# B&R Automation Studio project TD52 (part 76)

#### lib_properties.txt
```
For manual assignment to hardware configuration please
add the following additional include directories:

\Logical\MATLAB_includes\R2012b\

And the following additional build options:

-lm -D MODEL=LX2 -D NUMST=1 -D NCSTATES=0 -D HAVESTDIO -D ONESTEPFCN=1 -D TERMFCN=1 -D MAT_FILE=0 -D MULTI_INSTANCE_CODE=0 -D INTEGER_CODE=0 -D MT=0 -D CLASSIC_INTERFACE=0 -D TID01EQ=0
```

### Library Logical/EngineController/Lib_EC/lDAI (ANSIC, version 1.00.0) - Direct Air Injection 

#### DAI.c
```c
/********************************************************************
 * COPYRIGHT -- B&R Industrial Automation GmbH
 ********************************************************************
 * Program: DAI
 * File: DAI.c
 * Author: 105055527
 * Last modified by: cadm_kafkama00
 * Created: Sat Nov 11 23:05:34 2017
 * Last modified: Wed Oct 02 14:21:06 2024
 * Model Version: 4.14
 * Description: Direct Air Injection for J920 Faststart

   History:

   V0.02  Arnold, 27.11.2017,  tech demonstrator @ P20
   V0.03  Arnold, 24.10.2018,  rename from AirAss to DAI
   V0.04  Arnold, 24.10.2018,  deleted exhaust side DAI, deleted intake dynamics
   V0.05  Arnold, 14.08.2019,  unit testing done, pre-release for Pforzheim P21
   V0.06  Kafka, 20.09.2019, bug fix for testbench manual massflow testing
   V0.07  Kafka, 01.10.2019, massflow limitations changed from per valve to total massflow
   V0.08  Kafka, 02.10.2019, mass flow limitation over boost pressure removed for speed ramp
   V0.09  Kafka, 14.10.2019, disable for negative power trajectory is added in the enable subblock
   V0.10  Kafka, 18.12.2019, disable on speed hysteresis during speed ramp
   V4.14  Kafka, 06.09.2024, update to Matlab Version 2021b

 * modified Comment:
 ********************************************************************
 * Implementation of program DAI
 ********************************************************************
 * Generated with B&R Automation Studio Target for Simulink V6.7.1
 * (ERT based)
 ********************************************************************/

#include "DAI.h"
#include "DAI_private.h"

/*  Defines */

/*  Data Types */

/**************************** GLOBAL DATA *************************************/
/*  Definitions */

/*  Declarations  */

/* Forward declaration for local functions */
static void DAI_merge(int32_T idx[5], real32_T x[5], int32_T offset, int32_T np,
                      int32_T nq, int32_T iwork[5], real32_T xwork[5], struct fDAI* inst);
static void DAI_sort(real32_T x[5], int32_T idx[5], struct fDAI* inst);

/***************************** FILE SCOPE DATA ********************************/

/*************************** FUNCTIONS ****************************************/

/* Lookup Binary Search Utility BINARYSEARCH_real32_T */
void BINARYSEARCH_real32_T(uint32_T *piLeft, uint32_T *piRght, real32_T u, const
  real32_T *pData, uint32_T iHi, struct fDAI* inst)
{
  /* Find the location of current input value in the data table. */
  *piLeft = 0U;
  *piRght = iHi;
  if (u <= pData[0] ) {
    /* Less than or equal to the smallest point in the table. */
    *piRght = 0U;
  } else if (u >= pData[iHi] ) {
    /* Greater than or equal to the largest point in the table. */
    *piLeft = iHi;
  } else {
    uint32_T i;

    /* Do a binary search. */
    while (( *piRght - *piLeft ) > 1U ) {
      /* Get the average of the left and right indices using to Floor rounding. */
      i = (*piLeft + *piRght) >> 1;

      /* Move either the right index or the left index so that */
      /*  LeftDataPoint <= CurrentValue < RightDataPoint */
      if (u < pData[i] ) {
        *piRght = i;
      } else {
        *piLeft = i;
      }
    }
  }
}

/* Lookup Utility LookUp_real32_T_real32_T */
void LookUp_real32_T_real32_T(real32_T *pY, const real32_T *pYData, real32_T u,
  const real32_T *pUData, uint32_T iHi, struct fDAI* inst)
{
  uint32_T iLeft;
  uint32_T iRght;
  BINARYSEARCH_real32_T( &(iLeft), &(iRght), u, pUData, iHi, inst);

  {
    real32_T lambda;
    if (pUData[iRght] > pUData[iLeft] ) {
      real32_T num;
      real32_T den;
      den = pUData[iRght];
      den -= pUData[iLeft];
      num = u;
      num -= pUData[iLeft];
      lambda = num / den;
    } else {
      lambda = 0.0F;
    }

    {
      real32_T yLeftCast;
      real32_T yRghtCast;
      yLeftCast = pYData[iLeft];
      yRghtCast = pYData[iRght];
      yLeftCast += lambda * ( yRghtCast - yLeftCast );
      (*pY) = yLeftCast;
    }
  }
}

/*
 * Output and update for atomic system:
 *    '<S2>/Hystersis'
 *    '<S2>/Hystersis2'
 */
void DAI_Hystersis(real32_T rtu_Gw, real32_T rtu_Hy, real32_T rtu_In,
                   rtB_Hystersis_DAI *localB, rtDW_Hystersis_DAI *localDW, struct fDAI* inst)
{
  localDW->Inter = ((rtu_In >= rtu_Gw) || ((rtu_In >= rtu_Gw - rtu_Hy) &&
    localDW->Inter));
  localB->Out = localDW->Inter;
}

/* Function for MATLAB Function: '<S10>/MATLAB Function' */
static void DAI_merge(int32_T idx[5], real32_T x[5], int32_T offset, int32_T np,
                      int32_T nq, int32_T iwork[5], real32_T xwork[5], struct fDAI* inst)
{
  int32_T q;
  if ((np != 0) && (nq != 0)) {
    int32_T iout;
    int32_T n;
    int32_T n_tmp;
    n_tmp = np + nq;
    for (q = 0; q < n_tmp; q++) {
      iout = offset + q;
      iwork[q] = idx[iout];
      xwork[q] = x[iout];
    }

    n = 0;
    q = np;
    iout = offset - 1;
    int32_T exitg1;
    do {
      exitg1 = 0;
      iout++;
      if (xwork[n] <= xwork[q]) {
        idx[iout] = iwork[n];
        x[iout] = xwork[n];
        if (n + 1 < np) {
          n++;
        } else {
          exitg1 = 1;
        }
      } else {
        idx[iout] = iwork[q];
        x[iout] = xwork[q];
        if (q + 1 < n_tmp) {
          q++;
        } else {
          q = iout - n;
          while (n + 1 <= np) {
            iout = (q + n) + 1;
            idx[iout] = iwork[n];
            x[iout] = xwork[n];
            n++;
          }

          exitg1 = 1;
        }
      }
    } while (exitg1 == 0);
  }
}

/* Function for MATLAB Function: '<S10>/MATLAB Function' */
static void DAI_sort(real32_T x[5], int32_T idx[5], struct fDAI* inst)
{
  int32_T iwork[5];
  int32_T i2;
  int32_T i3;
  int32_T ib;
  int32_T k;
  real32_T xwork[5];
  real32_T x4[4];
  int8_T idx4[4];
  int8_T perm[4];
  x4[0] = 0.0F;
  idx4[0] = 0;
  x4[1] = 0.0F;
  idx4[1] = 0;
  x4[2] = 0.0F;
  idx4[2] = 0;
  x4[3] = 0.0F;
  idx4[3] = 0;
  ib = 0;
  for (k = 0; k < 5; k++) {
    idx[k] = 0;
    ib++;
    idx4[ib - 1] = (int8_T)(k + 1);
    x4[ib - 1] = x[k];
    if (ib == 4) {
      int32_T i4;
      real32_T tmp;
      real32_T tmp_0;
      if (x4[0] <= x4[1]) {
        ib = 1;
        i2 = 2;
      } else {
        ib = 2;
        i2 = 1;
      }

      if (x4[2] <= x4[3]) {
        i3 = 3;
        i4 = 4;
      } else {
        i3 = 4;
        i4 = 3;
      }

      tmp = x4[ib - 1];
      tmp_0 = x4[i3 - 1];
      if (tmp <= tmp_0) {
        tmp = x4[i2 - 1];
        if (tmp <= tmp_0) {
          perm[0] = (int8_T)ib;
          perm[1] = (int8_T)i2;
          perm[2] = (int8_T)i3;
          perm[3] = (int8_T)i4;
        } else if (tmp <= x4[i4 - 1]) {
          perm[0] = (int8_T)ib;
          perm[1] = (int8_T)i3;
          perm[2] = (int8_T)i2;
          perm[3] = (int8_T)i4;
        } else {
          perm[0] = (int8_T)ib;
          perm[1] = (int8_T)i3;
          perm[2] = (int8_T)i4;
          perm[3] = (int8_T)i2;
        }
      } else {
        tmp_0 = x4[i4 - 1];
        if (tmp <= tmp_0) {
          if (x4[i2 - 1] <= tmp_0) {
            perm[0] = (int8_T)i3;
            perm[1] = (int8_T)ib;
            perm[2] = (int8_T)i2;
            perm[3] = (int8_T)i4;
          } else {
            perm[0] = (int8_T)i3;
            perm[1] = (int8_T)ib;
            perm[2] = (int8_T)i4;
            perm[3] = (int8_T)i2;
          }
        } else {
          perm[0] = (int8_T)i3;
          perm[1] = (int8_T)i4;
          perm[2] = (int8_T)ib;
          perm[3] = (int8_T)i2;
        }
      }

      idx[k - 3] = idx4[perm[0] - 1];
      idx[k - 2] = idx4[perm[1] - 1];
      idx[k - 1] = idx4[perm[2] - 1];
      idx[k] = idx4[perm[3] - 1];
      x[k - 3] = x4[perm[0] - 1];
      x[k - 2] = x4[perm[1] - 1];
      x[k - 1] = x4[perm[2] - 1];
      x[k] = x4[perm[3] - 1];
      ib = 0;
    }
  }

  if (ib > 0) {
    perm[1] = 0;
    perm[2] = 0;
    perm[3] = 0;
    if (ib == 1) {
      perm[0] = 1;
    } else if (ib == 2) {
      if (x4[0] <= x4[1]) {
        perm[0] = 1;
        perm[1] = 2;
      } else {
        perm[0] = 2;
        perm[1] = 1;
      }
    } else if (x4[0] <= x4[1]) {
      if (x4[1] <= x4[2]) {
        perm[0] = 1;
        perm[1] = 2;
        perm[2] = 3;
      } else if (x4[0] <= x4[2]) {
        perm[0] = 1;
        perm[1] = 3;
        perm[2] = 2;
      } else {
        perm[0] = 3;
        perm[1] = 1;
        perm[2] = 2;
      }
    } else if (x4[0] <= x4[2]) {
      perm[0] = 2;
      perm[1] = 1;
      perm[2] = 3;
    } else if (x4[1] <= x4[2]) {
      perm[0] = 2;
      perm[1] = 3;
      perm[2] = 1;
    } else {
      perm[0] = 3;
      perm[1] = 2;
      perm[2] = 1;
    }

    for (k = 0; k < ib; k++) {
      i2 = perm[k] - 1;
      i3 = (k - ib) + 5;
      idx[i3] = idx4[i2];
      x[i3] = x4[i2];
    }
  }

  for (k = 0; k < 5; k++) {
    iwork[k] = 0;
    xwork[k] = 0.0F;
  }

  DAI_merge(idx, x, 0, 4, 1, iwork, xwork, inst);
}

/* Model step function */
void DAI_step(RT_MODEL_DAI *const DAI_M, struct fDAI* inst)
{
  struct BlockIO_DAI *DAI_B = DAI_M->blockIO;
  struct D_Work_DAI *DAI_DWork = DAI_M->dwork;

  /* local block i/o variables */
  real32_T rtb_CorrInternal[2];
  real32_T rtb_LookupTableDynamic2;
  real32_T rtb_LookupTableDynamic2_g;
  real32_T rtb_Saturation2[2];
  int32_T iidx[5];
  int32_T i;
  real32_T rtb_x_out[5];
  real32_T rtb_y_out[5];
  real32_T rtb_rCd[2];
  real32_T rtb_Disableintakedynamics1;
  real32_T rtb_Product_nc;
  real32_T rtb_Switch2_i;
  real32_T rtb_Switch2_n;
  real32_T rtb_UkYk1;
  real32_T rtb_rFlow_eng_act;
  real32_T rtb_rFlow_eng_des;
  boolean_T rtb_LogicalOperator2;
  boolean_T rtb_LogicalOperator5;

  /* S-Function (bur_bus_in): '<Root>/Bus Input3' */
  DAI_B->BusInput3 = inst->In;

  /* S-Function (bur_bus_in): '<Root>/Bus Input1' */
  DAI_B->BusInput1 = inst->Para;

  /* Outputs for Atomic SubSystem: '<Root>/EngineMassFlow' */
  /* MATLAB Function: '<S3>/desired engine massflow' incorporates:
   *  Constant: '<S27>/Constant1'
   *  MATLAB Function: '<S3>/actual engine massflow'
   *  Sum: '<S27>/Add1'
   */
  rtb_rFlow_eng_act = fmaxf((DAI_B->BusInput3.rT_T2s + 273.15F) * 287.15F, 1.0F);
  rtb_Disableintakedynamics1 = DAI_B->BusInput3.rVE_Eng *
    DAI_B->BusInput3.rV_EngDis;

  /* Outputs for Atomic SubSystem: '<Root>/Enable' */
  /* Product: '<S3>/Product' incorporates:
   *  Product: '<S2>/Product'
   */
  rtb_Product_nc = DAI_B->BusInput3.rN_Set_Norm * DAI_B->BusInput1.rN_EngNom;

  /* End of Outputs for SubSystem: '<Root>/Enable' */

  /* MATLAB Function: '<S3>/desired engine massflow' incorporates:
   *  Constant: '<S25>/Constant1'
   *  Constant: '<S30>/Constant1'
   *  Product: '<S25>/Product'
   *  Product: '<S30>/Product'
   *  Product: '<S3>/Product'
   */
  rtb_rFlow_eng_des = DAI_B->BusInput3.rPr_P2s_des * 100000.0F *
    rtb_Disableintakedynamics1 / rtb_rFlow_eng_act * (rtb_Product_nc *
    0.104719758F) / 2.0F / 6.28318548F;

  /* Switch: '<S23>/Switch2' incorporates:
   *  Constant: '<S3>/Constant4'
   *  RelationalOperator: '<S23>/LowerRelop1'
   *  RelationalOperator: '<S23>/UpperRelop'
   *  Switch: '<S23>/Switch'
   */
  if (DAI_B->BusInput3.rN_Eng > DAI_B->BusInput1.rN_EngNom) {
    rtb_Switch2_i = DAI_B->BusInput1.rN_EngNom;
  } else if (DAI_B->BusInput3.rN_Eng < 1.0F) {
    /* Switch: '<S23>/Switch' incorporates:
     *  Constant: '<S3>/Constant4'
     */
    rtb_Switch2_i = 1.0F;
  } else {
    rtb_Switch2_i = DAI_B->BusInput3.rN_Eng;
  }

  /* End of Switch: '<S23>/Switch2' */

  /* MATLAB Function: '<S3>/actual engine massflow' incorporates:
   *  Constant: '<S26>/Constant1'
   *  Constant: '<S29>/Constant1'
   *  Product: '<S26>/Product'
   *  Product: '<S29>/Product'
   */
  rtb_rFlow_eng_act = DAI_B->BusInput3.rPr_P2s_Avg * 100000.0F *
    rtb_Disableintakedynamics1 / rtb_rFlow_eng_act * (rtb_Switch2_i *
    0.104719758F) / 2.0F / 6.28318548F;

  /* End of Outputs for SubSystem: '<Root>/EngineMassFlow' */

  /* S-Function (bur_bus_in): '<Root>/Bus Input2' */
  DAI_B->BusInput2 = inst->Perm;

  /* Outputs for Atomic SubSystem: '<Root>/AirFlowDemand' */
  /* MATLAB Function: '<S10>/MATLAB Function' incorporates:
   *  Product: '<S10>/Divide'
   *  SignalConversion generated from: '<S13>/ SFunction '
   */
  rtb_x_out[0] = DAI_B->BusInput1.rN_DAI_On;
  rtb_x_out[1] = DAI_B->BusInput1.rN_EngNom * DAI_B->BusInput2.rNref_ff[0];
  rtb_x_out[2] = DAI_B->BusInput1.rN_EngNom * DAI_B->BusInput2.rNref_ff[1];
  rtb_x_out[3] = DAI_B->BusInput1.rN_EngNom * DAI_B->BusInput2.rNref_ff[2];
  rtb_x_out[4] = DAI_B->BusInput1.rN_DAI_Off;
  DAI_sort(rtb_x_out, iidx, inst);
  for (i = 0; i < 5; i++) {
    rtb_y_out[i] = DAI_B->BusInput2.rFlowRef_ff[iidx[i] - 1];
  }

  /* End of MATLAB Function: '<S10>/MATLAB Function' */

  /* Switch: '<S1>/ManMode' incorporates:
   *  Constant: '<S22>/Constant'
   *  Constant: '<S6>/Constant'
   *  RelationalOperator: '<S22>/Compare'
   *  RelationalOperator: '<S6>/Compare'
   *  Switch: '<S1>/OpMode'
   *  Switch: '<S3>/Disable intake dynamics1'
   */
  if (DAI_B->BusInput3.Test.bManEnable) {
    rtb_Disableintakedynamics1 = DAI_B->BusInput3.Test.rManMassReq;
  } else if (DAI_B->BusInput3.iOpMode <= 45) {
    /* S-Function (sfix_look1_dyn): '<S10>/Lookup Table Dynamic2' incorporates:
     *  Switch: '<S1>/OpMode'
     */
    /* Dynamic Look-Up Table Block: '<S10>/Lookup Table Dynamic2'
     * Input0  Data Type:  Floating Point real32_T
     * Input1  Data Type:  Floating Point real32_T
     * Input2  Data Type:  Floating Point real32_T
     * Output0 Data Type:  Floating Point real32_T
     * Lookup Method: Linear_Endpoint
     *
     */
    LookUp_real32_T_real32_T( &(rtb_LookupTableDynamic2_g), &rtb_y_out[0],
      DAI_B->BusInput3.rN_Eng, &rtb_x_out[0], 4U, inst);

    /* Switch: '<S1>/OpMode' incorporates:
     *  Product: '<S10>/Product3'
     */
    rtb_Disableintakedynamics1 = DAI_B->BusInput1.rGain_DAI_Start *
      rtb_LookupTableDynamic2_g;
  } else {
    /* Outputs for Atomic SubSystem: '<Root>/EngineMassFlow' */
    if (DAI_B->BusInput3.iOpMode < 50) {
      /* Switch: '<S3>/Disable intake dynamics1' incorporates:
       *  Constant: '<S3>/Constant1'
       */
      rtb_Switch2_i = 0.0F;
    } else {
      /* Switch: '<S3>/Disable intake dynamics1' incorporates:
       *  Sum: '<S3>/Add'
       */
      rtb_Switch2_i = rtb_rFlow_eng_des - rtb_rFlow_eng_act;
    }

    /* End of Outputs for SubSystem: '<Root>/EngineMassFlow' */

    /* Product: '<S1>/Product3' incorporates:
     *  Switch: '<S1>/OpMode'
     */
    rtb_Disableintakedynamics1 = rtb_Switch2_i * DAI_B->BusInput1.rGain_DAI;

    /* S-Function (sfix_look1_dyn): '<S1>/Lookup Table Dynamic2' incorporates:
     *  Switch: '<S1>/OpMode'
     */
    /* Dynamic Look-Up Table Block: '<S1>/Lookup Table Dynamic2'
     * Input0  Data Type:  Floating Point real32_T
     * Input1  Data Type:  Floating Point real32_T
     * Input2  Data Type:  Floating Point real32_T
     * Output0 Data Type:  Floating Point real32_T
     * Lookup Method: Linear_Endpoint
     *
     */
    LookUp_real32_T_real32_T( &(rtb_LookupTableDynamic2),
      &DAI_B->BusInput2.rRefFlowMaxP2s_y[0], DAI_B->BusInput3.rPr_P2s_Avg,
      &DAI_B->BusInput2.rRefFlowMaxP2s_x[0], 4U, inst);

    /* Switch: '<S8>/Switch2' incorporates:
     *  Constant: '<S1>/Constant2'
     *  RelationalOperator: '<S8>/LowerRelop1'
     *  RelationalOperator: '<S8>/UpperRelop'
     *  Switch: '<S1>/OpMode'
     *  Switch: '<S8>/Switch'
     */
    if (rtb_Disableintakedynamics1 > rtb_LookupTableDynamic2) {
      rtb_Disableintakedynamics1 = rtb_LookupTableDynamic2;
    } else if (rtb_Disableintakedynamics1 < 0.0F) {
      /* Switch: '<S8>/Switch' incorporates:
       *  Constant: '<S1>/Constant2'
       */
      rtb_Disableintakedynamics1 = 0.0F;
    }

    /* End of Switch: '<S8>/Switch2' */
  }

  /* End of Switch: '<S1>/ManMode' */

  /* Switch: '<S9>/Switch2' incorporates:
   *  Constant: '<S1>/Constant1'
   *  RelationalOperator: '<S9>/LowerRelop1'
   *  RelationalOperator: '<S9>/UpperRelop'
   *  Switch: '<S9>/Switch'
   */
  if (rtb_Disableintakedynamics1 > DAI_B->BusInput2.rMaxFlow) {
    rtb_Disableintakedynamics1 = DAI_B->BusInput2.rMaxFlow;
  } else if (rtb_Disableintakedynamics1 < 0.0F) {
    /* Switch: '<S9>/Switch' incorporates:
     *  Constant: '<S1>/Constant1'
     */
    rtb_Disableintakedynamics1 = 0.0F;
  }

  /* End of Switch: '<S9>/Switch2' */

  /* Abs: '<S7>/Abs' */
  rtb_Switch2_i = fabsf(DAI_B->BusInput2.rRateLimPos);

  /* Product: '<S11>/delta rise limit' incorporates:
   *  SampleTimeMath: '<S11>/sample time'
   *
   * About '<S11>/sample time':
   *  y = K where K = ( w * Ts )
   */
  rtb_Switch2_n = rtb_Switch2_i * 0.01F;

  /* Sum: '<S11>/Difference Inputs1' incorporates:
   *  UnitDelay: '<S11>/Delay Input2'
   */
  rtb_UkYk1 = rtb_Disableintakedynamics1 - DAI_DWork->DelayInput2_DSTATE;

  /* Switch: '<S12>/Switch2' incorporates:
   *  RelationalOperator: '<S12>/LowerRelop1'
   */
  if (rtb_UkYk1 <= rtb_Switch2_n) {
    /* Product: '<S11>/delta fall limit' incorporates:
     *  Abs: '<S7>/Abs1'
     *  Gain: '<S7>/Gain'
     *  SampleTimeMath: '<S11>/sample time'
     *
     * About '<S11>/sample time':
     *  y = K where K = ( w * Ts )
     */
    rtb_Switch2_n = -fabsf(DAI_B->BusInput2.rRateLimNeg) * 0.01F;

    /* Switch: '<S12>/Switch' incorporates:
     *  RelationalOperator: '<S12>/UpperRelop'
     */
    if (rtb_UkYk1 >= rtb_Switch2_n) {
      rtb_Switch2_n = rtb_UkYk1;
    }

    /* End of Switch: '<S12>/Switch' */
  }

  /* End of Switch: '<S12>/Switch2' */

  /* Sum: '<S11>/Difference Inputs2' incorporates:
   *  UnitDelay: '<S11>/Delay Input2'
   */
  rtb_UkYk1 = rtb_Switch2_n + DAI_DWork->DelayInput2_DSTATE;

  /* Switch: '<S7>/Rate limits selection' */
  if (rtb_Switch2_i >= 1.0E-6F) {
    rtb_Disableintakedynamics1 = rtb_UkYk1;
  }

  /* End of Switch: '<S7>/Rate limits selection' */

  /* Update for UnitDelay: '<S11>/Delay Input2' */
  DAI_DWork->DelayInput2_DSTATE = rtb_UkYk1;

  /* End of Outputs for SubSystem: '<Root>/AirFlowDemand' */

  /* Outputs for Atomic SubSystem: '<Root>/Enable' */
  /* Sum: '<S2>/Add' */
  rtb_Switch2_i = rtb_Product_nc - DAI_B->BusInput3.rN_Eng;

  /* MATLAB Function: '<S2>/Hystersis1' */
  DAI_DWork->Inter_n = ((rtb_Switch2_i >= DAI_B->BusInput2.rNDiffOn) ||
                        ((rtb_Switch2_i > DAI_B->BusInput2.rNDiffOff) &&
    DAI_DWork->Inter_n));

  /* MATLAB Function: '<S2>/Hystersis' */
  DAI_Hystersis(DAI_B->BusInput2.rFlowActOn, DAI_B->BusInput2.rFlowActHyst,
                rtb_Disableintakedynamics1, &DAI_B->sf_Hystersis,
                &DAI_DWork->sf_Hystersis, inst);

  /* MATLAB Function: '<S2>/Hystersis2' incorporates:
   *  Sum: '<S2>/Add1'
   */
  DAI_Hystersis(DAI_B->BusInput2.rPrDiffOn, DAI_B->BusInput2.rPrDiffHyst,
                DAI_B->BusInput3.rPr_DAI_In - DAI_B->BusInput3.rPr_P2s_Avg,
                &DAI_B->sf_Hystersis2, &DAI_DWork->sf_Hystersis2, inst);

  /* Sum: '<S14>/Diff' incorporates:
   *  UnitDelay: '<S14>/UD'
   */
  rtb_Switch2_i = DAI_B->BusInput3.rP_GEN2_Norm - DAI_DWork->UD_DSTATE;

  /* MATLAB Function: '<S2>/Hystersis3' incorporates:
   *  Constant: '<S2>/Constant'
   *  Constant: '<S2>/Constant1'
   */
  DAI_DWork->Inter = ((rtb_Switch2_i >= -1.0E-7) || ((rtb_Switch2_i >= -1.2E-7) &&
    DAI_DWork->Inter));

  /* Outputs for Atomic SubSystem: '<S2>/TON' */
  /* Logic: '<S20>/Logical Operator2' incorporates:
   *  Logic: '<S20>/Logical Operator3'
   */
  rtb_LogicalOperator2 = !DAI_B->BusInput3.bP_Set_reached;

  /* DiscreteIntegrator: '<S20>/Discrete-Time Integrator' incorporates:
   *  Logic: '<S20>/Logical Operator2'
   */
  if (rtb_LogicalOperator2 || (DAI_DWork->DiscreteTimeIntegrator_PrevRese != 0))
  {
    DAI_DWork->DiscreteTimeIntegrator_DSTATE = 0.0F;
  }

  /* RelationalOperator: '<S20>/Relational Operator' incorporates:
   *  DiscreteIntegrator: '<S20>/Discrete-Time Integrator'
   */
  rtb_LogicalOperator5 = (DAI_DWork->DiscreteTimeIntegrator_DSTATE >=
    DAI_B->BusInput2.rTi_P_Set_reached_delay);

  /* Update for DiscreteIntegrator: '<S20>/Discrete-Time Integrator' incorporates:
   *  DataTypeConversion: '<S21>/Conversion'
   *  Logic: '<S20>/Logical Operator'
   *  Logic: '<S20>/Logical Operator1'
   *  Logic: '<S20>/Logical Operator2'
   */
  if (!rtb_LogicalOperator2) {
    DAI_DWork->DiscreteTimeIntegrator_DSTATE += (real32_T)
      ((!rtb_LogicalOperator5) && DAI_B->BusInput3.bP_Set_reached) * 0.01F;
  }

  DAI_DWork->DiscreteTimeIntegrator_PrevRese = (int8_T)rtb_LogicalOperator2;

  /* End of Update for DiscreteIntegrator: '<S20>/Discrete-Time Integrator' */
  /* End of Outputs for SubSystem: '<S2>/TON' */

  /* MATLAB Function: '<S2>/MATLAB Function' incorporates:
   *  Logic: '<S20>/Logical Operator3'
   *  MATLAB Function: '<S2>/Hystersis1'
   *  MATLAB Function: '<S2>/Hystersis3'
   */
  switch (DAI_B->BusInput3.iOpMode) {
   case 30:
    rtb_LogicalOperator2 = (DAI_B->BusInput1.bDAI_Active_Start &&
      DAI_B->sf_Hystersis.Out && DAI_DWork->Inter_n && (DAI_B->BusInput3.rN_Eng >=
      DAI_B->BusInput1.rN_DAI_On) && (DAI_B->BusInput3.rN_Eng <
      DAI_B->BusInput1.rN_DAI_Off) && DAI_B->sf_Hystersis2.Out);
    DAI_DWork->bStart2Idle = true;
    DAI_B->BusCreator.bDAI_Tank_Pr_Ena = true;
    break;

   case 40:
    if (DAI_DWork->bStart2Idle && (DAI_B->BusInput3.rN_Eng <=
         DAI_B->BusInput1.rN_EngNom * 0.95F)) {
      rtb_LogicalOperator2 = (DAI_B->BusInput1.bDAI_Active_Start &&
        DAI_B->sf_Hystersis.Out && DAI_DWork->Inter_n &&
        (DAI_B->BusInput3.rN_Eng >= DAI_B->BusInput1.rN_DAI_On) &&
        (DAI_B->BusInput3.rN_Eng < DAI_B->BusInput1.rN_DAI_Off) &&
        DAI_B->sf_Hystersis2.Out);
    } else {
      rtb_LogicalOperator2 = false;
      DAI_DWork->bStart2Idle = false;
    }

    DAI_B->BusCreator.bDAI_Tank_Pr_Ena = true;
    break;

   case 50:
    /* Outputs for Atomic SubSystem: '<S2>/TON' */
    rtb_LogicalOperator2 = (((((!rtb_LogicalOperator5) || rtb_LogicalOperator2) &&
      DAI_B->BusInput1.bDAI_Active_PowRamp) || DAI_B->BusInput1.bDAI_Active_NetP)
      && DAI_B->sf_Hystersis.Out && DAI_B->sf_Hystersis2.Out && DAI_DWork->Inter);

    /* End of Outputs for SubSystem: '<S2>/TON' */
    DAI_B->BusCreator.bDAI_Tank_Pr_Ena =
      !DAI_B->BusInput3.bAMM_Pr_AirStarter_Tank_Lo;
    DAI_DWork->bStart2Idle = false;
    break;

   case 60:
    rtb_LogicalOperator2 = (DAI_B->BusInput1.bDAI_Active_Island &&
      DAI_B->sf_Hystersis.Out && DAI_DWork->Inter_n && DAI_B->sf_Hystersis2.Out);
    DAI_DWork->bStart2Idle = false;
    DAI_B->BusCreator.bDAI_Tank_Pr_Ena =
      !DAI_B->BusInput3.bAMM_Pr_AirStarter_Tank_Lo;
    break;

   default:
    rtb_LogicalOperator2 = false;
    DAI_DWork->bStart2Idle = false;
    DAI_B->BusCreator.bDAI_Tank_Pr_Ena = true;
    break;
  }

  /* End of MATLAB Function: '<S2>/MATLAB Function' */

  /* Logic: '<S2>/Logical Operator3' incorporates:
   *  Logic: '<S2>/Logical Operator2'
   */
  rtb_LogicalOperator2 = (DAI_B->BusInput1.bDAI_Active && (rtb_LogicalOperator2 &&
    DAI_B->BusInput3.bDAI_ena));

  /* Logic: '<S2>/Logical Operator4' incorporates:
   *  Logic: '<S2>/Logical Operator5'
   */
  DAI_B->BusCreator.bDAI_DP_Warn = (DAI_B->BusInput3.bDAI_ena &&
    (!DAI_B->sf_Hystersis2.Out));

  /* Update for UnitDelay: '<S14>/UD' */
  DAI_DWork->UD_DSTATE = DAI_B->BusInput3.rP_GEN2_Norm;

  /* End of Outputs for SubSystem: '<Root>/Enable' */

  /* Outputs for Atomic SubSystem: '<Root>/ValvePos' */
  /* Switch: '<S33>/Switch' incorporates:
   *  DataTypeConversion: '<S5>/Data Type Conversion'
   *  RelationalOperator: '<S33>/Relational Operator'
   */
  if (DAI_ConstB.Conversion >= DAI_B->BusInput2.iNumValve) {
    rtb_Switch2_i = DAI_ConstB.Conversion;
  } else {
    rtb_Switch2_i = DAI_B->BusInput2.iNumValve;
  }

  /* End of Switch: '<S33>/Switch' */

  /* Product: '<S5>/Product' */
  rtb_UkYk1 = 1.0F / rtb_Switch2_i * rtb_Disableintakedynamics1;

  /* Switch: '<S35>/Switch2' incorporates:
   *  Constant: '<S5>/Constant1'
   *  Constant: '<S5>/Constant3'
   *  RelationalOperator: '<S35>/LowerRelop1'
   *  RelationalOperator: '<S35>/UpperRelop'
   *  Switch: '<S35>/Switch'
   */
  if (DAI_B->BusInput3.rPr_DAI_A > 10.0F) {
    rtb_Switch2_i = 10.0F;
  } else if (DAI_B->BusInput3.rPr_DAI_A < 2.0F) {
    /* Switch: '<S35>/Switch' incorporates:
     *  Constant: '<S5>/Constant3'
     */
    rtb_Switch2_i = 2.0F;
  } else {
    rtb_Switch2_i = DAI_B->BusInput3.rPr_DAI_A;
  }

  /* End of Switch: '<S35>/Switch2' */

  /* Product: '<S37>/Product' incorporates:
   *  Constant: '<S37>/Constant1'
   */
  rtb_Product_nc = rtb_Switch2_i * 100000.0F;

  /* Product: '<S36>/Product' incorporates:
   *  Constant: '<S36>/Constant1'
   */
  rtb_Switch2_i = DAI_B->BusInput3.rPr_P2s_A * 100000.0F;

  /* MATLAB Function: '<S5>/Discharge coefficient computation_A' incorporates:
   *  Constant: '<S40>/Constant1'
   *  Sum: '<S40>/Add1'
   */
  if (rtb_Product_nc >= rtb_Switch2_i) {
    rtb_Switch2_i = fmaxf(rtb_Switch2_i / rtb_Product_nc, 1.0E-6F);
    if (rtb_Switch2_i >= 0.52828178771717416) {
      rtb_Switch2_i = sqrtf((powf(rtb_Switch2_i, 1.42857146F) - powf
        (rtb_Switch2_i, 1.71428573F)) * 3.5F);
    } else {
      rtb_Switch2_i = 0.484178245F;
    }

    rtb_Product_nc = rtb_UkYk1 / fmaxf(DAI_B->BusInput2.rDiam *
      DAI_B->BusInput2.rDiam * 3.14159274F / 4.0F * rtb_Product_nc * sqrtf(2.0F /
      fmaxf((DAI_B->BusInput3.rT_DAI + 273.15F) * 287.15F, 1.0E-6F)) *
      rtb_Switch2_i, 1.0E-6F);
  } else {
    rtb_Product_nc = 0.0F;
  }

  /* End of MATLAB Function: '<S5>/Discharge coefficient computation_A' */

  /* Switch: '<S34>/Switch2' incorporates:
   *  Constant: '<S5>/Constant4'
   *  Constant: '<S5>/Constant5'
   *  RelationalOperator: '<S34>/LowerRelop1'
   *  RelationalOperator: '<S34>/UpperRelop'
   *  Switch: '<S34>/Switch'
   */
  if (DAI_B->BusInput3.rPr_DAI_B > 10.0F) {
    rtb_Switch2_i = 10.0F;
  } else if (DAI_B->BusInput3.rPr_DAI_B < 2.0F) {
    /* Switch: '<S34>/Switch' incorporates:
     *  Constant: '<S5>/Constant5'
     */
    rtb_Switch2_i = 2.0F;
  } else {
    rtb_Switch2_i = DAI_B->BusInput3.rPr_DAI_B;
  }

  /* End of Switch: '<S34>/Switch2' */

  /* Product: '<S39>/Product' incorporates:
   *  Constant: '<S39>/Constant1'
   */
  rtb_Switch2_n = rtb_Switch2_i * 100000.0F;

  /* Product: '<S38>/Product' incorporates:
   *  Constant: '<S38>/Constant1'
   */
  rtb_Switch2_i = DAI_B->BusInput3.rPr_P2s_B * 100000.0F;

  /* MATLAB Function: '<S5>/Discharge coefficient computation_B' incorporates:
   *  Constant: '<S40>/Constant1'
   *  Sum: '<S40>/Add1'
   */
  if (rtb_Switch2_n >= rtb_Switch2_i) {
    rtb_Switch2_i = fmaxf(rtb_Switch2_i / rtb_Switch2_n, 1.0E-6F);
    if (rtb_Switch2_i >= 0.52828178771717416) {
      rtb_Switch2_i = sqrtf((powf(rtb_Switch2_i, 1.42857146F) - powf
        (rtb_Switch2_i, 1.71428573F)) * 3.5F);
    } else {
      rtb_Switch2_i = 0.484178245F;
    }

    rtb_Switch2_i = rtb_UkYk1 / fmaxf(DAI_B->BusInput2.rDiam *
      DAI_B->BusInput2.rDiam * 3.14159274F / 4.0F * rtb_Switch2_n * sqrtf(2.0F /
      fmaxf((DAI_B->BusInput3.rT_DAI + 273.15F) * 287.15F, 1.0E-6F)) *
      rtb_Switch2_i, 1.0E-6F);
  } else {
    rtb_Switch2_i = 0.0F;
  }

  /* End of MATLAB Function: '<S5>/Discharge coefficient computation_B' */

  /* Saturate: '<S5>/Saturation1' */
  if (rtb_Product_nc > 1.0F) {
    rtb_rCd[0] = 1.0F;
  } else if (rtb_Product_nc < 0.0F) {
    rtb_rCd[0] = 0.0F;
  } else {
    rtb_rCd[0] = rtb_Product_nc;
  }

  if (rtb_Switch2_i > 1.0F) {
    rtb_rCd[1] = 1.0F;
  } else if (rtb_Switch2_i < 0.0F) {
    rtb_rCd[1] = 0.0F;
  } else {
    rtb_rCd[1] = rtb_Switch2_i;
  }

  /* End of Saturate: '<S5>/Saturation1' */

  /* Switch: '<S5>/ManMode' */
  if (DAI_B->BusInput3.Test.bManPosEnable) {
    rtb_UkYk1 = DAI_B->BusInput3.Test.rManPos[0];
    rtb_Product_nc = DAI_B->BusInput3.Test.rManPos[1];
  } else {
    /* S-Function (sfix_look1_dyn): '<S5>/Cd2Pos' */
    /* Dynamic Look-Up Table Block: '<S5>/Cd2Pos'
     * Input0  Data Type:  Floating Point real32_T
     * Input1  Data Type:  Floating Point real32_T
     * Input2  Data Type:  Floating Point real32_T
     * Output0 Data Type:  Floating Point real32_T
     * Lookup Method: Linear_Endpoint
     *
     */
    LookUp_real32_T_real32_T( &(rtb_Saturation2[0]),
      &DAI_B->BusInput2.rPosBrkPts[0], rtb_rCd[0], &DAI_B->BusInput2.rDisBrkPts
      [0], 10U, inst);
    LookUp_real32_T_real32_T( &(rtb_Saturation2[1]),
      &DAI_B->BusInput2.rPosBrkPts[0], rtb_rCd[1], &DAI_B->BusInput2.rDisBrkPts
      [0], 10U, inst);

    /* Saturate: '<S5>/Saturation2' incorporates:
     *  Product: '<S5>/Product2'
     */
    rtb_Saturation2[0] *= DAI_B->BusInput2.rGainFlow;

    /* Saturate: '<S5>/Saturation2' */
    if (rtb_Saturation2[0] > 1.0F) {
      /* Saturate: '<S5>/Saturation2' */
      rtb_Saturation2[0] = 1.0F;
    } else if (rtb_Saturation2[0] < 0.0F) {
      /* Saturate: '<S5>/Saturation2' */
      rtb_Saturation2[0] = 0.0F;
    }

    /* Saturate: '<S5>/Saturation2' incorporates:
     *  Product: '<S5>/Product2'
     */
    rtb_Saturation2[1] *= DAI_B->BusInput2.rGainFlow;

    /* Saturate: '<S5>/Saturation2' */
    if (rtb_Saturation2[1] > 1.0F) {
      /* Saturate: '<S5>/Saturation2' */
      rtb_Saturation2[1] = 1.0F;
    } else if (rtb_Saturation2[1] < 0.0F) {
      /* Saturate: '<S5>/Saturation2' */
      rtb_Saturation2[1] = 0.0F;
    }

    /* S-Function (sfix_look1_dyn): '<S5>/CorrInternal' */
    /* Dynamic Look-Up Table Block: '<S5>/CorrInternal'
     * Input0  Data Type:  Floating Point real32_T
     * Input1  Data Type:  Floating Point real32_T
     * Input2  Data Type:  Floating Point real32_T
     * Output0 Data Type:  Floating Point real32_T
     * Lookup Method: Linear_Endpoint
     *
     */
    LookUp_real32_T_real32_T( &(rtb_CorrInternal[0]),
      &DAI_B->BusInput2.rRefValve_y[0], rtb_Saturation2[0],
      &DAI_B->BusInput2.rRefValve_x[0], 4U, inst);
    LookUp_real32_T_real32_T( &(rtb_CorrInternal[1]),
      &DAI_B->BusInput2.rRefValve_y[0], rtb_Saturation2[1],
      &DAI_B->BusInput2.rRefValve_x[0], 4U, inst);
    rtb_UkYk1 = rtb_CorrInternal[0];
    rtb_Product_nc = rtb_CorrInternal[1];
  }

  /* End of Switch: '<S5>/ManMode' */

  /* Logic: '<S5>/Logical Operator1' */
  rtb_LogicalOperator5 = (rtb_LogicalOperator2 ||
    DAI_B->BusInput3.Test.bManPosEnable);

  /* Saturate: '<S5>/Saturation3' */
  if (rtb_UkYk1 > 1.0F) {
    rtb_UkYk1 = 1.0F;
  } else if (rtb_UkYk1 < 0.0F) {
    rtb_UkYk1 = 0.0F;
  }

  /* Switch: '<S5>/Enable' */
  if (rtb_LogicalOperator5) {
    /* BusCreator: '<Root>/Bus Creator' */
    DAI_B->BusCreator.rPos_DAI_Set_A = rtb_UkYk1;
  } else {
    /* BusCreator: '<Root>/Bus Creator' incorporates:
     *  Constant: '<S5>/Constant2'
     */
    DAI_B->BusCreator.rPos_DAI_Set_A = 0.0F;
  }

  /* End of Outputs for SubSystem: '<Root>/ValvePos' */

  /* BusCreator: '<Root>/Bus Creator1' */
  DAI_B->BusCreator1.rPos_AirValve[0] = rtb_UkYk1;

  /* Outputs for Atomic SubSystem: '<Root>/ValvePos' */
  /* Saturate: '<S5>/Saturation3' */
  if (rtb_Product_nc > 1.0F) {
    rtb_UkYk1 = 1.0F;
  } else if (rtb_Product_nc < 0.0F) {
    rtb_UkYk1 = 0.0F;
  } else {
    rtb_UkYk1 = rtb_Product_nc;
  }

  /* Switch: '<S5>/Enable' */
  if (rtb_LogicalOperator5) {
    /* BusCreator: '<Root>/Bus Creator' */
    DAI_B->BusCreator.rPos_DAI_Set_B = rtb_UkYk1;
  } else {
    /* BusCreator: '<Root>/Bus Creator' incorporates:
     *  Constant: '<S5>/Constant2'
     */
    DAI_B->BusCreator.rPos_DAI_Set_B = 0.0F;
  }

  /* End of Outputs for SubSystem: '<Root>/ValvePos' */

  /* BusCreator: '<Root>/Bus Creator' */
  DAI_B->BusCreator.bDAI_V_Dem = rtb_LogicalOperator2;
  DAI_B->BusCreator.rFlow_DAI_Dem = rtb_Disableintakedynamics1;

  /* S-Function (bur_bus_out): '<Root>/Bus Output1' */
  inst->Out = DAI_B->BusCreator;

  /* BusCreator: '<Root>/Bus Creator1' */
  DAI_B->BusCreator1.rFlow_eng_des = rtb_rFlow_eng_des;
  DAI_B->BusCreator1.rFlow_eng_act = rtb_rFlow_eng_act;
  DAI_B->BusCreator1.rCd[0] = rtb_rCd[0];
  DAI_B->BusCreator1.rCd[1] = rtb_rCd[1];
  DAI_B->BusCreator1.rPos_AirValve[1] = rtb_UkYk1;

  /* S-Function (bur_bus_out): '<Root>/Bus Output2' */
  inst->dbg = DAI_B->BusCreator1;

  /* UnitDelay: '<S4>/Unit Delay' */
  DAI_B->UnitDelay = DAI_DWork->UnitDelay_DSTATE;

  /* S-Function (bur_out): '<Root>/Output1' */
  inst->Version = DAI_B->UnitDelay;

  /* Update for UnitDelay: '<S4>/Unit Delay' */
  DAI_DWork->UnitDelay_DSTATE = DAI_ConstB.DataTypeConversion3;
}

/* Model initialize function */
void DAI_initialize(RT_MODEL_DAI *const DAI_M, struct fDAI* inst)
{
  /* (no initialization code required) */
  UNUSED_PARAMETER(DAI_M);
}

/* Model terminate function */
void DAI_terminate(RT_MODEL_DAI *const DAI_M, struct fDAI* inst)
{
  /* (no terminate code required) */
  UNUSED_PARAMETER(DAI_M);
}

/*======================== TOOL VERSION INFORMATION ==========================*
 * MATLAB 9.11 (R2021b)14-May-2021                                            *
 * Simulink 10.4 (R2021b)14-May-2021                                          *
 * Simulink Coder 9.6 (R2021b)14-May-2021                                     *
 * Embedded Coder 7.7 (R2021b)14-May-2021                                     *
 * Stateflow 10.5 (R2021b)14-May-2021                                         *
 *============================================================================*/

/*======================= LICENSE IN USE INFORMATION =========================*
 * matlab                                                                     *
 * matlab_coder                                                               *
 * real-time_workshop                                                         *
 * rtw_embedded_coder                                                         *
 * simulink                                                                   *
 *============================================================================*/
```

#### DAI.h
```c
/********************************************************************
 * COPYRIGHT -- B&R Industrial Automation GmbH
 ********************************************************************
 * Program: DAI
 * File: DAI.h
 * Author: 105055527
 * Last modified by: cadm_kafkama00
 * Created: Sat Nov 11 23:05:34 2017
 * Last modified: Wed Oct 02 14:21:06 2024
 * Model Version: 4.14
 * Description: Direct Air Injection for J920 Faststart

   History:

   V0.02  Arnold, 27.11.2017,  tech demonstrator @ P20
   V0.03  Arnold, 24.10.2018,  rename from AirAss to DAI
   V0.04  Arnold, 24.10.2018,  deleted exhaust side DAI, deleted intake dynamics
   V0.05  Arnold, 14.08.2019,  unit testing done, pre-release for Pforzheim P21
   V0.06  Kafka, 20.09.2019, bug fix for testbench manual massflow testing
   V0.07  Kafka, 01.10.2019, massflow limitations changed from per valve to total massflow
   V0.08  Kafka, 02.10.2019, mass flow limitation over boost pressure removed for speed ramp
   V0.09  Kafka, 14.10.2019, disable for negative power trajectory is added in the enable subblock
   V0.10  Kafka, 18.12.2019, disable on speed hysteresis during speed ramp
   V4.14  Kafka, 06.09.2024, update to Matlab Version 2021b

 * modified Comment:
 ********************************************************************
 * Header for program DAI
 ********************************************************************
 * Generated with B&R Automation Studio Target for Simulink V6.7.1
 * (ERT based)
 ********************************************************************/

#ifndef RTW_HEADER_DAI_h_
#define RTW_HEADER_DAI_h_
#include <math.h>
#ifndef DAI_COMMON_INCLUDES_
#define DAI_COMMON_INCLUDES_
#include "rtwtypes.h"
#endif                                 /* DAI_COMMON_INCLUDES_ */

#include "DAI_types.h"
#include "lDAI.h"
/* Beginning of Dynamic TypeDefs: */
/* End of Dynamic TypeDefs: */
#ifndef MIN
#define MIN(a,b)	((a) < (b) ? (a) : (b))
#endif

#ifndef MAX
#define MAX(a,b)	((a) > (b) ? (a) : (b))
#endif

#ifndef AST_ROUND
#define AST_ROUND(x) ((x)>=0?(long long)((x)+0.5):(long long)((x)-0.5))
#endif

#include "rt_defines.h"

/* Macros for accessing real-time model data structure */
#ifndef rtmGetBlockIO
#define rtmGetBlockIO(rtm)             ((rtm)->blockIO)
#endif

#ifndef rtmSetBlockIO
#define rtmSetBlockIO(rtm, val)        ((rtm)->blockIO = (val))
#endif

#ifndef rtmGetRootDWork
#define rtmGetRootDWork(rtm)           ((rtm)->dwork)
#endif

#ifndef rtmSetRootDWork
#define rtmSetRootDWork(rtm, val)      ((rtm)->dwork = (val))
#endif

#ifndef rtmGetErrorStatus
#define rtmGetErrorStatus(rtm)         ((rtm)->errorStatus)
#endif

#ifndef rtmSetErrorStatus
#define rtmSetErrorStatus(rtm, val)    ((rtm)->errorStatus = (val))
#endif

#ifndef MIN
#define MIN(a,b)                       ((a) < (b) ? (a) : (b))
#endif

#ifndef MAX
#define MAX(a,b)                       ((a) > (b) ? (a) : (b))
#endif

#ifndef AST_ROUND
#define AST_ROUND(x)                   ((x)>=0?(long long)((x)+0.5):(long long)((x)-0.5))
#endif

/* user code (top of header file) */
/***************************************************************************************************
 * COPYRIGHT -- INNIO Jenbacher GmbH & CO OG
 ****************************************************************************************************
 * Program:            DAI
 * Author:             cadm_kafkama00
 * Created:            02.10.2024 14:21
 ****************************************************************************************************
 * MODEL INFORMATION
 ****************************************************************************************************
 * Model Name:         C:\Users\kafkama00\Documents\Git\DirectAirInjection\DAI.slx
 * Model Version:      4.14
 * Simulink Version:   R2021b
 * B&R Target:         V6.7.1
 * Description:        Direct Air Injection for J920 Faststart
 *
 *                     History:
 *
 *                        V0.02  Arnold, 27.11.2017,  tech demonstrator @ P20
 *                        V0.03  Arnold, 24.10.2018,  rename from AirAss to DAI
 *                        V0.04  Arnold, 24.10.2018,  deleted exhaust side DAI, deleted intake dynamics
 *                        V0.05  Arnold, 14.08.2019,  unit testing done, pre-release for Pforzheim P21
 *                        V0.06  Kafka, 20.09.2019, bug fix for testbench manual massflow testing
 *                        V0.07  Kafka, 01.10.2019, massflow limitations changed from per valve to total massflow
 *                        V0.08  Kafka, 02.10.2019, mass flow limitation over boost pressure removed for speed ramp
 *                        V0.09  Kafka, 14.10.2019, disable for negative power trajectory is added in the enable subblock
 *                        V0.10  Kafka, 18.12.2019, disable on speed hysteresis during speed ramp
 *                        V4.14  Kafka, 06.09.2024, update to Matlab Version 2021b
 *
 *
 ****************************************************************************************************
 * Last Modified By:   cadm_kafkama00
 * Last Modified Date: Wed Oct 02 14:20:47 2024
 ****************************************************************************************************/

/* Block signals for system '<S2>/Hystersis' */

/* Block states (default storage) for system '<S2>/Hystersis' */

/* Block signals (default storage) */

/* Block states (default storage) for system '<Root>' */

/* Invariant block signals (default storage) */

/* Real-time Model Data Structure */

extern const ConstBlockIO_DAI DAI_ConstB;/* constant block i/o */

/* Model entry point functions */
extern void DAI_initialize(RT_MODEL_DAI *const DAI_M, struct fDAI* inst);
extern void DAI_step(RT_MODEL_DAI *const DAI_M, struct fDAI* inst);
extern void DAI_terminate(RT_MODEL_DAI *const DAI_M, struct fDAI* inst);

/*-
 * The generated code includes comments that allow you to trace directly
 * back to the appropriate location in the model.  The basic format
 * is <system>/block_name, where system is the system number (uniquely
 * assigned by Simulink) and block_name is the name of the block.
 *
 * Use the MATLAB hilite_system command to trace the generated code back
 * to the model.  For example,
 *
 * hilite_system('<S3>')    - opens system 3
 * hilite_system('<S3>/Kp') - opens and selects block Kp which resides in S3
 *
 * Here is the system hierarchy for this model
 *
 * '<Root>' : 'DAI'
 * '<S1>'   : 'DAI/AirFlowDemand'
 * '<S2>'   : 'DAI/Enable'
 * '<S3>'   : 'DAI/EngineMassFlow'
 * '<S4>'   : 'DAI/Info'
 * '<S5>'   : 'DAI/ValvePos'
 * '<S6>'   : 'DAI/AirFlowDemand/Compare To Constant'
 * '<S7>'   : 'DAI/AirFlowDemand/RateLimit'
 * '<S8>'   : 'DAI/AirFlowDemand/Saturation Dynamic1'
 * '<S9>'   : 'DAI/AirFlowDemand/Saturation Dynamic2'
 * '<S10>'  : 'DAI/AirFlowDemand/SpeedRampMassFlow'
 * '<S11>'  : 'DAI/AirFlowDemand/RateLimit/Rate Limiter Dynamic'
 * '<S12>'  : 'DAI/AirFlowDemand/RateLimit/Rate Limiter Dynamic/Saturation Dynamic'
 * '<S13>'  : 'DAI/AirFlowDemand/SpeedRampMassFlow/MATLAB Function'
 * '<S14>'  : 'DAI/Enable/Difference'
 * '<S15>'  : 'DAI/Enable/Hystersis'
 * '<S16>'  : 'DAI/Enable/Hystersis1'
 * '<S17>'  : 'DAI/Enable/Hystersis2'
 * '<S18>'  : 'DAI/Enable/Hystersis3'
 * '<S19>'  : 'DAI/Enable/MATLAB Function'
 * '<S20>'  : 'DAI/Enable/TON'
 * '<S21>'  : 'DAI/Enable/TON/Data Type Conversion Inherited'
 * '<S22>'  : 'DAI/EngineMassFlow/Compare To Constant'
 * '<S23>'  : 'DAI/EngineMassFlow/Saturation Dynamic'
 * '<S24>'  : 'DAI/EngineMassFlow/actual engine massflow'
 * '<S25>'  : 'DAI/EngineMassFlow/bar2Pa'
 * '<S26>'  : 'DAI/EngineMassFlow/bar2Pa1'
 * '<S27>'  : 'DAI/EngineMassFlow/degC2K'
 * '<S28>'  : 'DAI/EngineMassFlow/desired engine massflow'
 * '<S29>'  : 'DAI/EngineMassFlow/rpm2rad'
 * '<S30>'  : 'DAI/EngineMassFlow/rpm2rad1'
 * '<S31>'  : 'DAI/ValvePos/Discharge coefficient computation_A'
 * '<S32>'  : 'DAI/ValvePos/Discharge coefficient computation_B'
 * '<S33>'  : 'DAI/ValvePos/Divisor'
 * '<S34>'  : 'DAI/ValvePos/Saturation Dynamic1'
 * '<S35>'  : 'DAI/ValvePos/Saturation Dynamic2'
 * '<S36>'  : 'DAI/ValvePos/bar2Pa'
 * '<S37>'  : 'DAI/ValvePos/bar2Pa1'
 * '<S38>'  : 'DAI/ValvePos/bar2Pa2'
 * '<S39>'  : 'DAI/ValvePos/bar2Pa3'
 * '<S40>'  : 'DAI/ValvePos/degC2K'
 * '<S41>'  : 'DAI/ValvePos/Divisor/Data Type Conversion Inherited'
 */
#endif                                 /* RTW_HEADER_DAI_h_ */
```

#### DAI_data.c
```c
/********************************************************************
 * COPYRIGHT -- B&R Industrial Automation GmbH
 ********************************************************************
 * Program: DAI
 * File: DAI_data.c
 * Author: 105055527
 * Last modified by: cadm_kafkama00
 * Created: Sat Nov 11 23:05:34 2017
 * Last modified: Wed Oct 02 14:21:06 2024
 * Model Version: 4.14
 * Description: Direct Air Injection for J920 Faststart

   History:

   V0.02  Arnold, 27.11.2017,  tech demonstrator @ P20
   V0.03  Arnold, 24.10.2018,  rename from AirAss to DAI
   V0.04  Arnold, 24.10.2018,  deleted exhaust side DAI, deleted intake dynamics
   V0.05  Arnold, 14.08.2019,  unit testing done, pre-release for Pforzheim P21
   V0.06  Kafka, 20.09.2019, bug fix for testbench manual massflow testing
   V0.07  Kafka, 01.10.2019, massflow limitations changed from per valve to total massflow
   V0.08  Kafka, 02.10.2019, mass flow limitation over boost pressure removed for speed ramp
   V0.09  Kafka, 14.10.2019, disable for negative power trajectory is added in the enable subblock
   V0.10  Kafka, 18.12.2019, disable on speed hysteresis during speed ramp
   V4.14  Kafka, 06.09.2024, update to Matlab Version 2021b

 * modified Comment:
 ********************************************************************
 * Data for program DAI
 ********************************************************************
 * Generated with B&R Automation Studio Target for Simulink V6.7.1
 * (ERT based)
 ********************************************************************/

#include "DAI.h"
#include "DAI_private.h"

/*  GLOBAL DATA DEFINITIONS */

/* Invariant block signals (default storage) */
const ConstBlockIO_DAI DAI_ConstB = {
  414U,                                /* '<S4>/Data Type Conversion3' */
  1.0F                                 /* '<S41>/Conversion' */
};
```

#### DAI_private.h
```c
/********************************************************************
 * COPYRIGHT -- B&R Industrial Automation GmbH
 ********************************************************************
 * Program: DAI
 * File: DAI_private.h
 * Author: 105055527
 * Last modified by: cadm_kafkama00
 * Created: Sat Nov 11 23:05:34 2017
 * Last modified: Wed Oct 02 14:21:06 2024
 * Model Version: 4.14
 * Description: Direct Air Injection for J920 Faststart

   History:

   V0.02  Arnold, 27.11.2017,  tech demonstrator @ P20
   V0.03  Arnold, 24.10.2018,  rename from AirAss to DAI
   V0.04  Arnold, 24.10.2018,  deleted exhaust side DAI, deleted intake dynamics
   V0.05  Arnold, 14.08.2019,  unit testing done, pre-release for Pforzheim P21
   V0.06  Kafka, 20.09.2019, bug fix for testbench manual massflow testing
   V0.07  Kafka, 01.10.2019, massflow limitations changed from per valve to total massflow
   V0.08  Kafka, 02.10.2019, mass flow limitation over boost pressure removed for speed ramp
   V0.09  Kafka, 14.10.2019, disable for negative power trajectory is added in the enable subblock
   V0.10  Kafka, 18.12.2019, disable on speed hysteresis during speed ramp
   V4.14  Kafka, 06.09.2024, update to Matlab Version 2021b

 * modified Comment:
 ********************************************************************
 * Header for program DAI
 ********************************************************************
 * Generated with B&R Automation Studio Target for Simulink V6.7.1
 * (ERT based)
 ********************************************************************/

#ifndef RTW_HEADER_DAI_private_h_
#define RTW_HEADER_DAI_private_h_
#include "rtwtypes.h"
#include "DAI.h"
#include <bur/plctypes.h>
#ifndef MIN
#define MIN(a,b)                       ((a) < (b) ? (a) : (b))
#endif

#ifndef MAX
#define MAX(a,b)                       ((a) > (b) ? (a) : (b))
#endif

#ifndef AST_ROUND
#define AST_ROUND(x)                   ((x)>=0?(long long)((x)+0.5):(long long)((x)-0.5))
#endif

void BINARYSEARCH_real32_T(uint32_T *piLeft, uint32_T *piRght, real32_T u, const
  real32_T *pData, uint32_T iHi, struct fDAI* inst);
void LookUp_real32_T_real32_T(real32_T *pY, const real32_T *pYData, real32_T u,
  const real32_T *pUData, uint32_T iHi, struct fDAI* inst);
extern void DAI_Hystersis(real32_T rtu_Gw, real32_T rtu_Hy, real32_T rtu_In,
  rtB_Hystersis_DAI *localB, rtDW_Hystersis_DAI *localDW, struct fDAI* inst);

#endif                                 /* RTW_HEADER_DAI_private_h_ */
```

#### DAI_types.h
```c
/********************************************************************
 * COPYRIGHT -- B&R Industrial Automation GmbH
 ********************************************************************
 * Program: DAI
 * File: DAI_types.h
 * Author: 105055527
 * Last modified by: cadm_kafkama00
 * Created: Sat Nov 11 23:05:34 2017
 * Last modified: Wed Oct 02 14:21:06 2024
 * Model Version: 4.14
 * Description: Direct Air Injection for J920 Faststart

   History:

   V0.02  Arnold, 27.11.2017,  tech demonstrator @ P20
   V0.03  Arnold, 24.10.2018,  rename from AirAss to DAI
   V0.04  Arnold, 24.10.2018,  deleted exhaust side DAI, deleted intake dynamics
   V0.05  Arnold, 14.08.2019,  unit testing done, pre-release for Pforzheim P21
   V0.06  Kafka, 20.09.2019, bug fix for testbench manual massflow testing
   V0.07  Kafka, 01.10.2019, massflow limitations changed from per valve to total massflow
   V0.08  Kafka, 02.10.2019, mass flow limitation over boost pressure removed for speed ramp
   V0.09  Kafka, 14.10.2019, disable for negative power trajectory is added in the enable subblock
   V0.10  Kafka, 18.12.2019, disable on speed hysteresis during speed ramp
   V4.14  Kafka, 06.09.2024, update to Matlab Version 2021b

 * modified Comment:
 ********************************************************************
 * Header for program DAI
 ********************************************************************
 * Generated with B&R Automation Studio Target for Simulink V6.7.1
 * (ERT based)
 ********************************************************************/

#ifndef RTW_HEADER_DAI_types_h_
#define RTW_HEADER_DAI_types_h_
#include "rtwtypes.h"

/* Model Code Variants */
#ifndef MIN
#define MIN(a,b)                       ((a) < (b) ? (a) : (b))
#endif

#ifndef MAX
#define MAX(a,b)                       ((a) > (b) ? (a) : (b))
#endif

#ifndef AST_ROUND
#define AST_ROUND(x)                   ((x)>=0?(long long)((x)+0.5):(long long)((x)-0.5))
#endif

/* Forward declaration for rtModel */

#endif                                 /* RTW_HEADER_DAI_types_h_ */
```

#### fDAI.c
```c
/********************************************************************
 * COPYRIGHT -- B&R Industrial Automation GmbH
 ********************************************************************
 * Program: DAI
 * File: fDAI.c
 * Author: 105055527
 * Last modified by: cadm_kafkama00
 * Created: Sat Nov 11 23:05:34 2017
 * Last modified: Wed Oct 02 14:21:06 2024
 * Model Version: 4.14
 * Description: Direct Air Injection for J920 Faststart

   History:

   V0.02  Arnold, 27.11.2017,  tech demonstrator @ P20
   V0.03  Arnold, 24.10.2018,  rename from AirAss to DAI
   V0.04  Arnold, 24.10.2018,  deleted exhaust side DAI, deleted intake dynamics
   V0.05  Arnold, 14.08.2019,  unit testing done, pre-release for Pforzheim P21
   V0.06  Kafka, 20.09.2019, bug fix for testbench manual massflow testing
   V0.07  Kafka, 01.10.2019, massflow limitations changed from per valve to total massflow
   V0.08  Kafka, 02.10.2019, mass flow limitation over boost pressure removed for speed ramp
   V0.09  Kafka, 14.10.2019, disable for negative power trajectory is added in the enable subblock
   V0.10  Kafka, 18.12.2019, disable on speed hysteresis during speed ramp
   V4.14  Kafka, 06.09.2024, update to Matlab Version 2021b

 * modified Comment:
 ********************************************************************
 * Implementation of program DAI
 ********************************************************************
 * Generated with B&R Automation Studio Target for Simulink V6.7.1
 * (ERT based)
 ********************************************************************/

#include <bur/plctypes.h>
#include "DAI.h"
#include "rtwtypes.h"

/* Defines */
#define SS_TERMINATE 4
#define SS_OUTPUT 3
#define SS_INITIALIZE 2

/*  Data Types */

/**************************** GLOBAL DATA *************************************/
/*  Definitions */

/*  Declarations  */

/***************************** FILE SCOPE DATA ********************************/

/*************************** FUNCTIONS ****************************************/
#ifdef __cplusplus

unsigned long bur_heap_size = 6553500;

#endif

/*LEGACYMODE_VARIABLES*/
void fDAI(struct fDAI* inst)
{
  tag_RTM_DAI* const DAI_M = &(inst)->bur_DAI;
	inst->bur_DAI.blockIO = &(inst)->bur_BlockIO_DAI;
	inst->bur_DAI.dwork = &(inst)->bur_D_Work_DAI;

  switch (inst->ssMethodType)
  {
   case SS_INITIALIZE:
    /* call model initialize function */
    DAI_initialize(DAI_M, inst);
    break;

   case SS_OUTPUT:
    /* call model step function */
    DAI_step(DAI_M, inst);

    break;

   case SS_TERMINATE:
    /* call model terminate function */
    DAI_terminate(DAI_M, inst);
    break;
  }
}

/*****************************************************************************
   Function block sample time: 0.01s
 *****************************************************************************/

/*****************************************************************************
   B&R Automation Studio Target for Simulink Version: A6.7.1 (02-Dec-2022)
 *****************************************************************************/

/*======================== TOOL VERSION INFORMATION ==========================*
 * MATLAB 9.11 (R2021b)14-May-2021                                            *
 * Simulink 10.4 (R2021b)14-May-2021                                          *
 * Simulink Coder 9.6 (R2021b)14-May-2021                                     *
 * Embedded Coder 7.7 (R2021b)14-May-2021                                     *
 * Stateflow 10.5 (R2021b)14-May-2021                                         *
 *============================================================================*/

/*======================= LICENSE IN USE INFORMATION =========================*
 * matlab                                                                     *
 * matlab_coder                                                               *
 * real-time_workshop                                                         *
 * rtw_embedded_coder                                                         *
 * simulink                                                                   *
 *============================================================================*/
```

#### lDAI.fun
```iecst
FUNCTION_BLOCK fDAI
  VAR_INPUT
    ssMethodType: SINT;
  END_VAR
  VAR_INPUT
        In : DAI_In_Bus; (**)
  END_VAR
  VAR_INPUT
        Para : DAI_Para_Bus; (**)
  END_VAR
  VAR_INPUT
        Perm : DAI_Perm_Bus; (**)
  END_VAR
  VAR_OUTPUT
        Out : DAI_Out_Bus; (**)
  END_VAR
  VAR_OUTPUT
        dbg : DAI_Dbg_Bus; (**)
  END_VAR
  VAR_OUTPUT
        Version : UDINT := 0; (**)
  END_VAR
	VAR
		bur_BlockIO_DAI : BlockIO_DAI;
	END_VAR
	VAR
		bur_D_Work_DAI : D_Work_DAI;
	END_VAR
	VAR
		bur_DAI : tag_RTM_DAI;
	END_VAR
END_FUNCTION_BLOCK
```

#### lDAI.typ
```iecst
TYPE
	DAI_Dbg_Bus :  STRUCT
		rFlow_eng_des :  REAL; (*Desired engine mass flow (kg/s)*)
		rFlow_eng_act :  REAL; (*Actual engine mass flow (kg/s)*)
		rCd :  ARRAY[0..1] OF REAL; (*Cd value (-)*)
		rPos_AirValve :  ARRAY[0..1] OF REAL; (*Position air valve (%)*)
	END_STRUCT;

	DAI_In_Bus :  STRUCT
		rPr_P2s_A :  REAL; (*Boost pressure bank A (bar)*)
		rPr_P2s_B :  REAL; (*Boost pressure bank B (bar)*)
		rPr_P2s_Avg :  REAL; (*Boost pressure average (bar)*)
		rPr_P2s_des :  REAL; (*Desired boost pressure (Gen2) (bar)*)
		rT_T2s :  REAL; (*Intake manifold temperature (degC)*)
		rPr_DAI_In :  REAL; (*air pressure upstream shut off valve (bar)*)
		rPr_DAI_A :  REAL; (*air pressure upstream control valve bank A (bar)*)
		rPr_DAI_B :  REAL; (*air pressure upstream control valve bank B (bar)*)
		rT_DAI :  REAL; (*air temperature upstream of control valves (degC)*)
		rN_Eng :  REAL; (*Engine speed (rpm)*)
		rN_Set_Norm :  REAL; (*Engine speed setpoint normalized (-)*)
		rV_EngDis :  REAL; (*Engine displacement (m3)*)
		rVE_Eng :  REAL; (*Volumetric efficiency (-)*)
		iOpMode :  INT; (*Operation mode (-)*)
		bP_Set_reached :  BOOL; (*target load reached (-)*)
		bDAI_ena :  BOOL; (*DAI enabled (-)*)
		Test :  DAI_Test_Bus; (*Testing inputs (-)*)
		bAMM_Pr_AirStarter_Tank_Lo :  BOOL; (*warning starter tank pressure low trigger (-)*)
		rP_GEN2_Norm :  REAL; (*normed Power trajectory from GEN2 (-)*)
	END_STRUCT;

	DAI_Out_Bus :  STRUCT
		rPos_DAI_Set_A :  REAL; (*Position air assist control valve bank A (pu)*)
		rPos_DAI_Set_B :  REAL; (*Position air assist control valve bank B (pu)*)
		bDAI_V_Dem :  BOOL; (*open (true) DAI slamshut valve (-)*)
		bDAI_Tank_Pr_Ena :  BOOL; (*starter tank pressure DAI enable (-)*)
		bDAI_DP_Warn :  BOOL; (*pressure difference DAI warning (-)*)
		rFlow_DAI_Dem :  REAL; (*demanded DAI air mass flow  (-)*)
	END_STRUCT;

	DAI_Para_Bus :  STRUCT
		rN_EngNom :  REAL; (*Nominal engine speed (rpm)*)
		bDAI_Active :  BOOL; (*Activate intake assist part (-)*)
		bDAI_Active_Start :  BOOL; (*DAI active during speed ramp (-)*)
		bDAI_Active_PowRamp :  BOOL; (*DAI active during load ramp (-)*)
		bDAI_Active_NetP :  BOOL; (*DAI active in grid mode (-)*)
		bDAI_Active_Island :  BOOL; (*DAI active in isolated mode (-)*)
		rN_DAI_On :  REAL; (*Engine speed to activate DAI during speed ramp  (rpm)*)
		rN_DAI_Off :  REAL; (*Engine speed to deactivate DAI during speed ramp  (rpm)*)
		rGain_DAI_Start :  REAL; (*DAI gain mass flow speed ramp (-)*)
		rGain_DAI :  REAL; (*DAI gain mass flow (-)*)
	END_STRUCT;

	DAI_Perm_Bus :  STRUCT
		rMaxFlow :  REAL; (*Max mass flow request air assist (kg/s)*)
		rRateLimPos :  REAL; (*Rate limitation of the air mass request, 0 no rate limit (kg/s/s)*)
		rRateLimNeg :  REAL; (*Rate limitation of the air mass request (kg/s/s)*)
		rDiam :  REAL; (*Diameter of DAI control valve (m)*)
		iNumValve :  USINT; (*Number of DAI control valves (-)*)
		rGainFlow :  REAL; (*Gain at output of valve position request (-)*)
		rDisBrkPts :  ARRAY[0..10] OF REAL; (*Discharge coeff breakpoints DAI control valve (-)*)
		rPosBrkPts :  ARRAY[0..10] OF REAL; (*Position breakpoints  DAI control valve (%)*)
		rFlowActOn :  REAL; (*Mass flow request to enable DAI (kg/s)*)
		rFlowActHyst :  REAL; (*Mass flow request to enable DAI hysteresis (kg/s)*)
		rNDiffOff :  REAL; (*Speed deviation request to enable DAI (rpm)*)
		rNDiffOn :  REAL; (*Speed deviation request to disable DAI (rpm)*)
		rPrDiffHyst :  REAL; (*pressure difference  to enable DAI hysteresis (bar)*)
		rPrDiffOn :  REAL; (*pressure difference  to enable DAI (bar)*)
		rRefValve_x :  ARRAY[0..4] OF REAL; (*Valve Position correction x-value (pu)*)
		rRefValve_y :  ARRAY[0..4] OF REAL; (*Valve Position correction y-value (pu)*)
		rNref_ff :  ARRAY[0..2] OF REAL; (*feed forward during speed ramp, speed normalized (x) (pu)*)
		rFlowRef_ff :  ARRAY[0..4] OF REAL; (*feed forward during speed ramp, flow (y) (kg/s)*)
		rRefFlowMaxP2s_x :  ARRAY[0..4] OF REAL; (*Maxmum mass flow based on p2s (x) (bar)*)
		rRefFlowMaxP2s_y :  ARRAY[0..4] OF REAL; (*Maxmum mass flow based on p2s (y) (kg/s)*)
		rTi_P_Set_reached_delay :  REAL; (*time delay after target load reached (s)*)
	END_STRUCT;

	DAI_Test_Bus :  STRUCT
		bManEnable :  BOOL; (*Enable manual mode (-)*)
		rManMassReq :  REAL; (*Manual air mass request (kg/s)*)
		bManPosEnable :  BOOL; (*Enable manual position mode (-)*)
		rManPos :  ARRAY[0..1] OF REAL; (*Manual air assist position (pu)*)
	END_STRUCT;

END_TYPE

TYPE
rtB_Hystersis_DAI : STRUCT
	Out : BOOL;
END_STRUCT;
rtDW_Hystersis_DAI : STRUCT
	Inter : BOOL;
END_STRUCT;
BlockIO_DAI : STRUCT
	BusInput2 : DAI_Perm_Bus;
	BusInput3 : DAI_In_Bus;
	BusInput1 : DAI_Para_Bus;
	BusCreator1 : DAI_Dbg_Bus;
	BusCreator : DAI_Out_Bus;
	UnitDelay : UDINT;
	sf_Hystersis2 : rtB_Hystersis_DAI;
	sf_Hystersis : rtB_Hystersis_DAI;
END_STRUCT;
D_Work_DAI : STRUCT
	UD_DSTATE : REAL;
	DiscreteTimeIntegrator_DSTATE : REAL;
	DelayInput2_DSTATE : REAL;
	UnitDelay_DSTATE : UDINT;
	DiscreteTimeIntegrator_PrevRese : SINT;
	bStart2Idle : BOOL;
	Inter : BOOL;
	Inter_n : BOOL;
	sf_Hystersis2 : rtDW_Hystersis_DAI;
	sf_Hystersis : rtDW_Hystersis_DAI;
END_STRUCT;
ConstBlockIO_DAI : STRUCT
	DataTypeConversion3 : UDINT;
	Conversion : REAL;
END_STRUCT;
tag_RTM_DAI : STRUCT
	errorStatus : REFERENCE TO USINT;
	blockIO : REFERENCE TO BlockIO_DAI;
	dwork : REFERENCE TO D_Work_DAI;
END_STRUCT;
RT_MODEL_DAI : tag_RTM_DAI;

END_TYPE
TYPE
END_TYPE
```

#### lib_properties.txt
```
For manual assignment to hardware configuration please
add the following additional include directories:

\Logical\MATLAB_includes\R2021b\

And the following additional build options:

-lm -D MODEL=DAI -D NUMST=1 -D NCSTATES=0 -D HAVESTDIO -D MODEL_HAS_DYNAMICALLY_LOADED_SFCNS=0 -D CLASSIC_INTERFACE=0 -D ALLOCATIONFCN=0 -D TID01EQ=0 -D TERMFCN=1 -D ONESTEPFCN=1 -D MAT_FILE=0 -D MULTI_INSTANCE_CODE=1 -D INTEGER_CODE=0 -D MT=0
```

#### rt_defines.h
```c
/********************************************************************
 * COPYRIGHT -- B&R Industrial Automation GmbH
 ********************************************************************
 * Program: DAI
 * File: rt_defines.h
 * Author: 105055527
 * Last modified by: cadm_kafkama00
 * Created: Sat Nov 11 23:05:34 2017
 * Last modified: Wed Oct 02 14:21:06 2024
 * Model Version: 4.14
 * Description: Direct Air Injection for J920 Faststart

   History:

   V0.02  Arnold, 27.11.2017,  tech demonstrator @ P20
   V0.03  Arnold, 24.10.2018,  rename from AirAss to DAI
   V0.04  Arnold, 24.10.2018,  deleted exhaust side DAI, deleted intake dynamics
   V0.05  Arnold, 14.08.2019,  unit testing done, pre-release for Pforzheim P21
   V0.06  Kafka, 20.09.2019, bug fix for testbench manual massflow testing
   V0.07  Kafka, 01.10.2019, massflow limitations changed from per valve to total massflow
   V0.08  Kafka, 02.10.2019, mass flow limitation over boost pressure removed for speed ramp
   V0.09  Kafka, 14.10.2019, disable for negative power trajectory is added in the enable subblock
   V0.10  Kafka, 18.12.2019, disable on speed hysteresis during speed ramp
   V4.14  Kafka, 06.09.2024, update to Matlab Version 2021b

 * modified Comment:
 ********************************************************************
 * Header for program DAI
 ********************************************************************
 * Generated with B&R Automation Studio Target for Simulink V6.7.1
 * (ERT based)
 ********************************************************************/

#ifndef RTW_HEADER_rt_defines_h_
#define RTW_HEADER_rt_defines_h_
#ifndef MIN
#define MIN(a,b)                       ((a) < (b) ? (a) : (b))
#endif

#ifndef MAX
#define MAX(a,b)                       ((a) > (b) ? (a) : (b))
#endif

#ifndef AST_ROUND
#define AST_ROUND(x)                   ((x)>=0?(long long)((x)+0.5):(long long)((x)-0.5))
#endif

/*===========*
 * Constants *
 *===========*/
#define RT_PI                          3.14159265358979323846
#define RT_PIF                         3.1415927F
#define RT_LN_10                       2.30258509299404568402
#define RT_LN_10F                      2.3025851F
#define RT_LOG10E                      0.43429448190325182765
#define RT_LOG10EF                     0.43429449F
#define RT_E                           2.7182818284590452354
#define RT_EF                          2.7182817F

/*
 * UNUSED_PARAMETER(x)
 *   Used to specify that a function parameter (argument) is required but not
 *   accessed by the function body.
 */
#ifndef UNUSED_PARAMETER
#if defined(__LCC__)
#define UNUSED_PARAMETER(x)                                      /* do nothing */
#else

/*
 * This is the semi-ANSI standard way of indicating that an
 * unused function parameter is required.
 */
#define UNUSED_PARAMETER(x)            (void) (x)
#endif
#endif
#endif                                 /* RTW_HEADER_rt_defines_h_ */
```

#### rtwtypes.h
```c
/********************************************************************
 * COPYRIGHT -- B&R Industrial Automation GmbH
 ********************************************************************
 * Program: DAI
 * File: rtwtypes.h
 * Author: 105055527
 * Last modified by: cadm_kafkama00
 * Created: Sat Nov 11 23:05:34 2017
 * Last modified: Wed Oct 02 14:21:06 2024
 * Model Version: 4.14
 * Description: Direct Air Injection for J920 Faststart

   History:

   V0.02  Arnold, 27.11.2017,  tech demonstrator @ P20
   V0.03  Arnold, 24.10.2018,  rename from AirAss to DAI
   V0.04  Arnold, 24.10.2018,  deleted exhaust side DAI, deleted intake dynamics
   V0.05  Arnold, 14.08.2019,  unit testing done, pre-release for Pforzheim P21
   V0.06  Kafka, 20.09.2019, bug fix for testbench manual massflow testing
   V0.07  Kafka, 01.10.2019, massflow limitations changed from per valve to total massflow
   V0.08  Kafka, 02.10.2019, mass flow limitation over boost pressure removed for speed ramp
   V0.09  Kafka, 14.10.2019, disable for negative power trajectory is added in the enable subblock
   V0.10  Kafka, 18.12.2019, disable on speed hysteresis during speed ramp
   V4.14  Kafka, 06.09.2024, update to Matlab Version 2021b

 * modified Comment:
 ********************************************************************
 * Header for program DAI
 ********************************************************************
 * Generated with B&R Automation Studio Target for Simulink V6.7.1
 * (ERT based)
 ********************************************************************/

#ifndef RTWTYPES_H
#define RTWTYPES_H

/* Logical type definitions */
#if (!defined(__cplusplus))
#ifndef false
#define false                          (0U)
#endif

#ifndef true
#define true                           (1U)
#endif
#endif

/*=======================================================================*
 * Target hardware information
 *   Device type: Intel->x86/Pentium
 *   Number of bits:     char:   8    short:   16    long:  32
 *                       long:  32
 *                       native word size:  32
 *   Byte ordering: LittleEndian
 *   Signed integer division rounds to: Zero
 *   Shift right on a signed integer as arithmetic shift: on
 *=======================================================================*/

/*=======================================================================*
 * Fixed width word size data types:                                     *
 *   int8_T, int16_T, int32_T     - signed 8, 16, or 32 bit integers     *
 *   uint8_T, uint16_T, uint32_T  - unsigned 8, 16, or 32 bit integers   *
 *   real32_T, real64_T           - 32 and 64 bit floating point numbers *
 *=======================================================================*/
typedef signed char int8_T;
typedef unsigned char uint8_T;
typedef short int16_T;
typedef unsigned short uint16_T;
typedef long int32_T;
typedef unsigned long uint32_T;
typedef float real32_T;
typedef double real64_T;

/*===========================================================================*
 * Generic type definitions: boolean_T, char_T, byte_T, int_T, uint_T,       *
 *                           real_T, time_T, ulong_T.                        *
 *===========================================================================*/
typedef double real_T;
typedef double time_T;
typedef unsigned char boolean_T;
typedef long int_T;
typedef unsigned long uint_T;
typedef unsigned long ulong_T;
typedef char char_T;
typedef unsigned char uchar_T;
typedef char_T byte_T;

/*=======================================================================*
 * Min and Max:                                                          *
 *   int8_T, int16_T, int32_T     - signed 8, 16, or 32 bit integers     *
 *   uint8_T, uint16_T, uint32_T  - unsigned 8, 16, or 32 bit integers   *
 *=======================================================================*/
#define MAX_int8_T                     ((int8_T)(127))
#define MIN_int8_T                     ((int8_T)(-128))
#define MAX_uint8_T                    ((uint8_T)(255U))
#define MAX_int16_T                    ((int16_T)(32767))
#define MIN_int16_T                    ((int16_T)(-32768))
#define MAX_uint16_T                   ((uint16_T)(65535U))
#define MAX_int32_T                    ((int32_T)(2147483647))
#define MIN_int32_T                    ((int32_T)(-2147483647-1))
#define MAX_uint32_T                   ((uint32_T)(0xFFFFFFFFU))

/* Block D-Work pointer type */
typedef void * pointer_T;

#endif                                 /* RTWTYPES_H */

#ifndef MIN
#define MIN(a,b)                       ((a) < (b) ? (a) : (b))
#endif

#ifndef MAX
#define MAX(a,b)                       ((a) > (b) ? (a) : (b))
#endif

#ifndef AST_ROUND
#define AST_ROUND(x)                   ((x)>=0?(long long)((x)+0.5):(long long)((x)-0.5))
#endif
```

### Library Logical/EngineController/Lib_EC/lTExhMon (ANSIC)

#### lTExhMon.fun
```iecst
FUNCTION_BLOCK fTExhMon
  VAR_INPUT
    ssMethodType: SINT;
  END_VAR  VAR_INPUT
        Para : tTExhMon_PARA; (**)
  END_VAR
  VAR_INPUT
        In : tTExhMon_IN; (**)
  END_VAR
 VAR_OUTPUT
        Out : tTExhMon_OUT; (**)
  END_VAR
 VAR_OUTPUT
        Dbg : tTExhMon_DBG; (**)
  END_VAR
  VAR_OUTPUT
        Version : UDINT; (**)
  END_VAR
	VAR
		bur_BlockIO_TExhMon : BlockIO_TExhMon;
	END_VAR
	VAR
		bur_D_Work_TExhMon : D_Work_TExhMon;
	END_VAR
	VAR
		bur_PrevZCSigStates_TExhMon : PrevZCSigStates_TExhMon;
	END_VAR
	VAR
		bur_ExternalOutputs_TExhMon : ExternalOutputs_TExhMon;
	END_VAR
END_FUNCTION_BLOCK
```

#### lTExhMon.typ
```iecst
TYPE

   tTExhMon_DBG : STRUCT
        rP_Act_Norm_Filt_dbg : REAL; (*Normalized power (-)*)
        rdT2Ref : ARRAY[0..24] OF REAL; (*Reference exhaust gas temperature (T_EPU - T_median) (°C)*)
        rT_EPU_EG_Cyl_Vect : ARRAY[0..24] OF REAL; (*Engine power unit exhaust gas temperature considering valid cylinders (°C)*)
        rCA_Ign_Act_Vect : ARRAY[0..24] OF REAL; (*Actual ignition timing point considering valid cylinders (°CA)*)
        rdT_Ref_Max_Cyl : ARRAY[0..24] OF REAL; (*Threshold depending on narrowed temperature monitoring (°C)*)
        bValidCyl : ARRAY[0..24] OF BOOL; (*Vector indicating valid cylinders for monitoring (-)*)
        bEGTSignalJump : ARRAY[0..24] OF BOOL; (*Vector indicating exhaust gas temperature signal jumps (-)*)
    END_STRUCT;

   tTExhMon_IN : STRUCT
        ucNumCyl : USINT; (*Total number of cylinders (-)*)
        bTExh_Mon_UseNarrowWindow : ARRAY[0..24] OF BOOL; (*narrower threshold activation for exhaust temperature monitoring (-)*)
        tGCB_On_Di : BOOL; (*generator circuit breaker closed (-)*)
        rT_EPU_EG : ARRAY[0..24] OF REAL; (*Exhaust Temperature per cylinder (°C)*)
        rP_Act_Norm_Filt : REAL; (*Actual power (-)*)
        rCA_Ign_Act : ARRAY[0..24] OF REAL; (*actual cylinder ignition point (°CA)*)
        rCA_IgnP_Set : REAL; (*ignition timing setpoint (°CA)*)
        rdTExh_Misfire : REAL; (*delta temperature from reference to misfire limit (°C)*)
        rT_dTExhMon_ITPComp : REAL; (*TExh compensation at later ITP values (positive values for increasing temp. at retarding) (K/°CA)*)
        MSAGT : ARRAY[0..24] OF BOOL; (*TExh sensor failure (-)*)
        rTs_task : REAL; (*Task sampling time (-)*)
    END_STRUCT;

   tTExhMon_OUT : STRUCT
        bdTExhMonTrip : ARRAY[0..24] OF BOOL; (*TRUE = TExhMon trip detected for cylinder (-)*)
        rT_Exh_Exp : ARRAY[0..24] OF REAL; (*expected temperature per cylinder (°C)*)
        rT_EG_Lim_dTExhMon : ARRAY[0..24] OF REAL; (*Trip Limit per cylinder (°C)*)
        rdT2Limit : ARRAY[0..24] OF REAL; (*current deviation from expected value per cylinder (°C)*)
        rdT2Limit_Max : ARRAY[0..24] OF REAL; (*MAX deviation since last engine start per cylinder (°C)*)
        rdT2Limit_Min : ARRAY[0..24] OF REAL; (*MIN deviation since last engine start per cylinder (°C)*)
        bdTExhMonTrip_all : BOOL; (*collection of alarm activation for all cylinders (-)*)
        bdTExhMon_Act : BOOL; (*TRUE = dTExhMon activated and running (-)*)
        rTExh_median : REAL; (*Exh Temp median (°C)*)
    END_STRUCT;

   tTExhMon_PARA : STRUCT
        tDelay_dTExhMon_Act : REAL; (*delay for activation of dTExhMon after GCB_ON (s)*)
        rdT_Ref_Max : REAL; (*distance from expected temperature to trip (normal) (°C)*)
        rFiltTau_Texh : REAL; (*constant for reference value filtering (s)*)
        rdT2Exp_Max : REAL; (*Max distance from expected value to trip limit (°C)*)
        tDelay_dTExhMon_Act_P : REAL; (*delay for re-activation after low power operation (s)*)
        bTExhMon_Release : BOOL; (*parameter that activates this function (s)*)
        rTExhBound_SensScal : REAL; (*Sensitivity scaling factor for the exhaust gas temperature tolerance boundary/range (-)*)
    END_STRUCT;
END_TYPE
TYPE
rtB_TON_TExhMon_Act_GCB_ON_TExh : STRUCT
	LogicalOperator3 : BOOL;
END_STRUCT;
rtDW_TON_TExhMon_Act_GCB_ON_TEx : STRUCT
	DiscreteTimeIntegrator_DSTATE : REAL;
	DiscreteTimeIntegrator_PrevRese : SINT;
END_STRUCT;
rtB_TON_InBound_TExhMon : STRUCT
	LogicalOperator3 : ARRAY[0..24] OF BOOL;
END_STRUCT;
rtDW_TON_InBound_TExhMon : STRUCT
	DiscreteTimeIntegrator_DSTATE : ARRAY[0..24] OF REAL;
	DiscreteTimeIntegrator_PrevRese : ARRAY[0..24] OF SINT;
END_STRUCT;
BlockIO_TExhMon : STRUCT
	BusInput : tTExhMon_IN;
	BusInput1 : tTExhMon_PARA;
	UnitDelay : UDINT;
	TON_OutBound : rtB_TON_InBound_TExhMon;
	TON_InBound : rtB_TON_InBound_TExhMon;
	xTON_bdTExhMon_Act_P : rtB_TON_TExhMon_Act_GCB_ON_TExh;
	TON_TExhMon_Act_GCB_ON : rtB_TON_TExhMon_Act_GCB_ON_TExh;
END_STRUCT;
D_Work_TExhMon : STRUCT
	Delay_DSTATE : ARRAY[0..24] OF REAL;
	Delay1_DSTATE : ARRAY[0..24] OF REAL;
	Delay2_DSTATE : ARRAY[0..24] OF REAL;
	DiscreteTimeIntegrator_DSTATE : ARRAY[0..24] OF REAL;
	UnitDelay_DSTATE : UDINT;
	rdT2Ref_1 : ARRAY[0..24] OF REAL;
	rCA_ITPOffset_1 : ARRAY[0..24] OF REAL;
	UnitDelay_DSTATE_i : ARRAY[0..24] OF BOOL;
	DelayInput1_DSTATE : ARRAY[0..24] OF BOOL;
	DiscreteTimeIntegrator_PrevRese : ARRAY[0..24] OF SINT;
	DiscreteTimeIntegrator_IC_LOADI : USINT;
	Memory_PreviousInput : BOOL;
	Memory_PreviousInput_o : BOOL;
	rdT2Ref_1_not_empty : BOOL;
	rCA_ITPOffset_1_not_empty : BOOL;
	bReset_1 : BOOL;
	TexhJump : ARRAY[0..24] OF BOOL;
	TON_OutBound : rtDW_TON_InBound_TExhMon;
	TON_InBound : rtDW_TON_InBound_TExhMon;
	xTON_bdTExhMon_Act_P : rtDW_TON_TExhMon_Act_GCB_ON_TEx;
	TON_TExhMon_Act_GCB_ON : rtDW_TON_TExhMon_Act_GCB_ON_TEx;
END_STRUCT;
PrevZCSigStates_TExhMon : STRUCT
	Delay1_Reset_ZCE : USINT;
	Delay2_Reset_ZCE : USINT;
END_STRUCT;
ConstParam_TExhMon : STRUCT
	pooled12 : ARRAY[0..15] OF BOOL;
END_STRUCT;
ExternalInputs_TExhMon : STRUCT
	In_TExhMon : tTExhMon_IN;
	Para_TExhMon : tTExhMon_PARA;
END_STRUCT;
ExternalOutputs_TExhMon : STRUCT
	Out : tTExhMon_OUT;
	Dbg : tTExhMon_DBG;
END_STRUCT;
END_TYPE
```

#### TExhMon.h
```c
/********************************************************************
 * COPYRIGHT -- Bernecker + Rainer Industrie-Elektronik Ges.m.b.H.
 ********************************************************************
 * Program: TExhMon
 * File: TExhMon.h
 * Author: 120011115
 * Created: Mon Sep 05 16:14:57 2016
 ********************************************************************
 * Header for program TExhMon
 ********************************************************************
 * Generated with B&R Automation Studio Target for Simulink V4.2
 * (ERT based)
 ********************************************************************/

#ifndef RTW_HEADER_TExhMon_h_
#define RTW_HEADER_TExhMon_h_
#ifndef TExhMon_COMMON_INCLUDES_
# define TExhMon_COMMON_INCLUDES_
#include <math.h>
#include "rtwtypes.h"
#endif                                 /* TExhMon_COMMON_INCLUDES_ */

#include "TExhMon_types.h"
#include "lTExhMon.h"

/* Macros for accessing real-time model data structure */
#ifndef rtmGetErrorStatus
# define rtmGetErrorStatus(rtm)        ((void*) 0)
#endif

#ifndef rtmSetErrorStatus
# define rtmSetErrorStatus(rtm, val)   ((void) 0)
#endif

#ifndef rtmGetStopRequested
# define rtmGetStopRequested(rtm)      ((void*) 0)
#endif

#ifndef MIN
#define MIN(a,b)                       ((a) < (b) ? (a) : (b))
#endif

#ifndef MAX
#define MAX(a,b)                       ((a) > (b) ? (a) : (b))
#endif

/* user code (top of header file) */
/***************************************************************************************************
 * COPYRIGHT -- INNIO Jenbacher GmbH & CO OG
 ****************************************************************************************************
 * Program:            TExhMon
 * Author:             schmisi00
 * Created:            12.01.2021 16:31
 ****************************************************************************************************
 * MODEL INFORMATION
 ****************************************************************************************************
 * Model Name:         c:\Git\ValveFractureMonitoring\EC_TExh_Monitoring\TExhMon.slx
 * Model Version:      1.05
 * Simulink Version:   R2012b
 * B&R Target:         V4.5.1
 * Description:        Exhaust Temperature Monitoring Function.
 *
 *                     Outstandings:
 *                     -------------
 *                     - NA
 ****************************************************************************************************
 * HISTORY
 ****************************************************************************************************
 * Last Modified By:   schmisi00
 * Last Modified Date: Tue Jan 12 16:15:42 2021
 * Modified Comment:   V1.00  20.10.2019 -  Created, model implementation from AS to Simulink
 *                     V1.01  20.11.2019 -  Added exhaust gas temperature tolerance range
 *                     V1.02  21.11.2019 -  Model cleanup, removed unused parameters and inputs
 *                     V1.03  10.12.2019 -  Bugfix, included number of cylinders in median calculation
 *                     V1.04  31.01.2020 -  Bugfix, corrected rdT2ref calculation when re-activation of invalid cylinders,
 *                                                      changed upper limit of parameter tDelay_dTExhMon_Act_Lim
 *                     V1.05  07.01.2020 -  Detection of exhaust gas temperature signal jumps
 ****************************************************************************************************/

/* Block signals for system '<S1>/TON_TExhMon_Act_GCB_ON' */

/* Block states (auto storage) for system '<S1>/TON_TExhMon_Act_GCB_ON' */

/* Block signals for system '<S5>/TON_InBound' */

/* Block states (auto storage) for system '<S5>/TON_InBound' */

/* Block signals (auto storage) */

/* Block states (auto storage) for system '<Root>' */

/* Zero-crossing (trigger) state */

/* Constant parameters (auto storage) */

/* External inputs (root inport signals with auto storage) */

/* External outputs (root outports fed by signals with auto storage) */

/* Constant parameters (auto storage) */
extern const ConstParam_TExhMon TExhMon_ConstP;

/* Model entry point functions */
extern void TExhMon_initialize(D_Work_TExhMon *TExhMon_DWork,
  PrevZCSigStates_TExhMon *TExhMon_PrevZCSigState, struct fTExhMon* inst);
extern void TExhMon_step(BlockIO_TExhMon *TExhMon_B, D_Work_TExhMon
  *TExhMon_DWork, PrevZCSigStates_TExhMon *TExhMon_PrevZCSigState,
  ExternalOutputs_TExhMon *TExhMon_Y, struct fTExhMon* inst);
extern void TExhMon_terminate(struct fTExhMon* inst);

/*-
 * The generated code includes comments that allow you to trace directly
 * back to the appropriate location in the model.  The basic format
 * is <system>/block_name, where system is the system number (uniquely
 * assigned by Simulink) and block_name is the name of the block.
 *
 * Use the MATLAB hilite_system command to trace the generated code back
 * to the model.  For example,
 *
 * hilite_system('<S3>')    - opens system 3
 * hilite_system('<S3>/Kp') - opens and selects block Kp which resides in S3
 *
 * Here is the system hierarchy for this model
 *
 * '<Root>' : 'TExhMon'
 * '<S1>'   : 'TExhMon/Activation Criterias'
 * '<S2>'   : 'TExhMon/Environment Controller'
 * '<S3>'   : 'TExhMon/Environment Controller1'
 * '<S4>'   : 'TExhMon/Info'
 * '<S5>'   : 'TExhMon/Init_Calculations'
 * '<S6>'   : 'TExhMon/PARA_Limitation'
 * '<S7>'   : 'TExhMon/TExh Mon Cont Exec'
 * '<S8>'   : 'TExhMon/Activation Criterias/S-R Flip-Flop'
 * '<S9>'   : 'TExhMon/Activation Criterias/S-R Flip-Flop1'
 * '<S10>'  : 'TExhMon/Activation Criterias/TON_TExhMon_Act_GCB_ON'
 * '<S11>'  : 'TExhMon/Activation Criterias/xTON_bdTExhMon_Act_P'
 * '<S12>'  : 'TExhMon/Activation Criterias/TON_TExhMon_Act_GCB_ON/Data Type Conversion Inherited'
 * '<S13>'  : 'TExhMon/Activation Criterias/xTON_bdTExhMon_Act_P/Data Type Conversion Inherited'
 * '<S14>'  : 'TExhMon/Init_Calculations/  '
 * '<S15>'  : 'TExhMon/Init_Calculations/  1'
 * '<S16>'  : 'TExhMon/Init_Calculations/EGT_SignalJumpDetection'
 * '<S17>'  : 'TExhMon/Init_Calculations/MATLAB Function'
 * '<S18>'  : 'TExhMon/Init_Calculations/TON_InBound'
 * '<S19>'  : 'TExhMon/Init_Calculations/TON_OutBound'
 * '<S20>'  : 'TExhMon/Init_Calculations/EGT_SignalJumpDetection/MATLAB Function1'
 * '<S21>'  : 'TExhMon/Init_Calculations/EGT_SignalJumpDetection/TOF'
 * '<S22>'  : 'TExhMon/Init_Calculations/EGT_SignalJumpDetection/TOF/Data Type Conversion Inherited'
 * '<S23>'  : 'TExhMon/Init_Calculations/TON_InBound/Data Type Conversion Inherited'
 * '<S24>'  : 'TExhMon/Init_Calculations/TON_OutBound/Data Type Conversion Inherited'
 * '<S25>'  : 'TExhMon/TExh Mon Cont Exec/Detect Increase'
 * '<S26>'  : 'TExhMon/TExh Mon Cont Exec/MATLAB Function'
 */
#endif                                 /* RTW_HEADER_TExhMon_h_ */
```

#### TExhMon_private.h
```c
/********************************************************************
 * COPYRIGHT -- Bernecker + Rainer Industrie-Elektronik Ges.m.b.H.
 ********************************************************************
 * Program: TExhMon
 * File: TExhMon_private.h
 * Author: 120011115
 * Created: Mon Sep 05 16:14:57 2016
 ********************************************************************
 * Header for program TExhMon
 ********************************************************************
 * Generated with B&R Automation Studio Target for Simulink V4.2
 * (ERT based)
 ********************************************************************/

#ifndef RTW_HEADER_TExhMon_private_h_
#define RTW_HEADER_TExhMon_private_h_
#include "rtwtypes.h"
#include <bur/plctypes.h>
#ifndef __RTWTYPES_H__
#error This file requires rtwtypes.h to be included
#else
#ifdef TMWTYPES_PREVIOUSLY_INCLUDED
#error This file requires rtwtypes.h to be included before tmwtypes.h
#else

/* Check for inclusion of an incorrect version of rtwtypes.h */
#ifndef RTWTYPES_ID_C08S16I32L32N32F1
#error This code was generated with a different "rtwtypes.h" than the file included
#endif                                 /* RTWTYPES_ID_C08S16I32L32N32F1 */
#endif                                 /* TMWTYPES_PREVIOUSLY_INCLUDED */
#endif                                 /* __RTWTYPES_H__ */

#ifndef MIN
#define MIN(a,b)                       ((a) < (b) ? (a) : (b))
#endif

#ifndef MAX
#define MAX(a,b)                       ((a) > (b) ? (a) : (b))
#endif

extern void TExhMon_TON_TExhMon_Act_GCB_ON(boolean_T rtu_IN, real32_T rtu_PT,
  rtB_TON_TExhMon_Act_GCB_ON_TExh *localB, rtDW_TON_TExhMon_Act_GCB_ON_TEx
  *localDW, struct fTExhMon* inst);
extern void TExhMon_TON_InBound(const boolean_T rtu_IN[25], real32_T rtu_PT,
  rtB_TON_InBound_TExhMon *localB, rtDW_TON_InBound_TExhMon *localDW, struct fTExhMon* inst);

#endif                                 /* RTW_HEADER_TExhMon_private_h_ */
```

#### TExhMon_types.h
```c
/********************************************************************
 * COPYRIGHT -- Bernecker + Rainer Industrie-Elektronik Ges.m.b.H.
 ********************************************************************
 * Program: TExhMon
 * File: TExhMon_types.h
 * Author: 120011115
 * Created: Mon Sep 05 16:14:57 2016
 ********************************************************************
 * Header for program TExhMon
 ********************************************************************
 * Generated with B&R Automation Studio Target for Simulink V4.2
 * (ERT based)
 ********************************************************************/

#ifndef RTW_HEADER_TExhMon_types_h_
#define RTW_HEADER_TExhMon_types_h_
#include "rtwtypes.h"
#ifndef MIN
#define MIN(a,b)                       ((a) < (b) ? (a) : (b))
#endif

#ifndef MAX
#define MAX(a,b)                       ((a) > (b) ? (a) : (b))
#endif

#ifndef _DEFINED_TYPEDEF_FOR_tTExhMon_PARA_Lim_
#define _DEFINED_TYPEDEF_FOR_tTExhMon_PARA_Lim_

typedef struct {
  real32_T tDelay_dTExhMon_Act_Lim;
  real32_T rdT_Ref_Max_Lim;
  real32_T rFiltTau_TExh_Lim;
  real32_T rdT2Exp_Max_Lim;
  real32_T tDelay_dTExhMon_Act_P_Lim;
  real32_T rTExhBound_SensScal_Lim;
} tTExhMon_PARA_Lim;

#endif
#endif                                 /* RTW_HEADER_TExhMon_types_h_ */
```

#### rtwtypes.h
```c
/********************************************************************
 * COPYRIGHT -- Bernecker + Rainer Industrie-Elektronik Ges.m.b.H.
 ********************************************************************
 * Program: TExhMon
 * File: rtwtypes.h
 * Author: 120011115
 * Created: Mon Sep 05 16:14:57 2016
 ********************************************************************
 * Header for program TExhMon
 ********************************************************************
 * Generated with B&R Automation Studio Target for Simulink V4.2
 * (ERT based)
 ********************************************************************/

#ifndef __RTWTYPES_H__
#define __RTWTYPES_H__
#ifndef TRUE
# define TRUE                          (1U)
#endif

#ifndef FALSE
# define FALSE                         (0U)
#endif

#ifndef __TMWTYPES__
#define __TMWTYPES__
#include <limits.h>

/*=======================================================================*
 * Target hardware information
 *   Device type: Intel->x86/Pentium
 *   Number of bits:     char:   8    short:   16    long:  32
 *                       long:  32
 *                       native word size:  32
 *   Byte ordering: LittleEndian
 *   Signed integer division rounds to: Zero
 *   Shift right on a signed integer as arithmetic shift: on
 *=======================================================================*/

/*=======================================================================*
 * Fixed width word size data types:                                     *
 *   int8_T, int16_T, int32_T     - signed 8, 16, or 32 bit integers     *
 *   uint8_T, uint16_T, uint32_T  - unsigned 8, 16, or 32 bit integers   *
 *   real32_T, real64_T           - 32 and 64 bit floating point numbers *
 *=======================================================================*/
typedef signed char int8_T;
typedef unsigned char uint8_T;
typedef short int16_T;
typedef unsigned short uint16_T;
typedef long int32_T;
typedef unsigned long uint32_T;
typedef float real32_T;
typedef double real64_T;

/*===========================================================================*
 * Generic type definitions: real_T, time_T, boolean_T, int_T, uint_T,       *
 *                           ulong_T, char_T and byte_T.                     *
 *===========================================================================*/
typedef double real_T;
typedef double time_T;
typedef unsigned char boolean_T;
typedef long int_T;
typedef unsigned long uint_T;
typedef unsigned long ulong_T;
typedef char char_T;
typedef unsigned char uchar_T;
typedef char_T byte_T;

/*=======================================================================*
 * Min and Max:                                                          *
 *   int8_T, int16_T, int32_T     - signed 8, 16, or 32 bit integers     *
 *   uint8_T, uint16_T, uint32_T  - unsigned 8, 16, or 32 bit integers   *
 *=======================================================================*/
#define MAX_int8_T                     ((int8_T)(127))
#define MIN_int8_T                     ((int8_T)(-128))
#define MAX_uint8_T                    ((uint8_T)(255U))
#define MIN_uint8_T                    ((uint8_T)(0U))
#define MAX_int16_T                    ((int16_T)(32767))
#define MIN_int16_T                    ((int16_T)(-32768))
#define MAX_uint16_T                   ((uint16_T)(65535U))
#define MIN_uint16_T                   ((uint16_T)(0U))
#define MAX_int32_T                    ((int32_T)(2147483647))
#define MIN_int32_T                    ((int32_T)(-2147483647-1))
#define MAX_uint32_T                   ((uint32_T)(0xFFFFFFFFU))
#define MIN_uint32_T                   ((uint32_T)(0U))

/* Logical type definitions */
#if (!defined(__cplusplus)) && (!defined(__true_false_are_keywords))
#  ifndef false
#   define false                       (0U)
#  endif

#  ifndef true
#   define true                        (1U)
#  endif
#endif

/*
 * Simulink Coder assumes the code is compiled on a target using a 2's complement representation
 * for signed integer values.
 */
#if ((SCHAR_MIN + 1) != -SCHAR_MAX)
#error "This code must be compiled using a 2's complement representation for signed integer values"
#endif

/* This ID is used to detect inclusion of an incompatible rtwtypes.h */
#define RTWTYPES_ID_C08S16I32L32N32F1
#else                                  /* __TMWTYPES__ */
#define TMWTYPES_PREVIOUSLY_INCLUDED
#endif                                 /* __TMWTYPES__ */

/* Block D-Work pointer type */
typedef void * pointer_T;

/* Simulink specific types */
#ifndef __SIMSTRUC_TYPES_H__
#define __SIMSTRUC_TYPES_H__

/* Trigger directions: falling, either, and rising */
typedef enum {
  FALLING_ZERO_CROSSING = -1,
  ANY_ZERO_CROSSING = 0,
  RISING_ZERO_CROSSING = 1
} ZCDirection;

/* Previous state of a trigger signal */
typedef uint8_T ZCSigState;

/* Initial value of a trigger zero crossing signal */
#define UNINITIALIZED_ZCSIG            0x03U
#define NEG_ZCSIG                      0x02U
#define POS_ZCSIG                      0x01U
#define ZERO_ZCSIG                     0x00U

/* Current state of a trigger signal */
typedef enum {
  FALLING_ZCEVENT = -1,
  NO_ZCEVENT = 0,
  RISING_ZCEVENT = 1
} ZCEventType;

#endif                                 /* __SIMSTRUC_TYPES_H__ */
#endif                                 /* __RTWTYPES_H__ */

#ifndef MIN
#define MIN(a,b)                       ((a) < (b) ? (a) : (b))
#endif

#ifndef MAX
#define MAX(a,b)                       ((a) > (b) ? (a) : (b))
#endif
```
